LIN {X 0,Y 573.225,Z 559.074,A -85,B 0,C 180,E1 -2028.544,E2 -2028.544} C_VEL
LIN {X 0,Y 573.245,Z 559.083,A -85,B 0,C 180,E1 -2031.3,E2 -2031.3} C_VEL
LIN {X 0,Y 573.262,Z 559.073,A -85,B 0,C 180,E1 -2034.012,E2 -2034.012} C_VEL
LIN {X 0,Y 573.284,Z 559.068,A -85,B 0,C 180,E1 -2036.52,E2 -2036.52} C_VEL
LIN {X 0,Y 573.227,Z 559.08,A -85,B 0,C 180,E1 -2039.119,E2 -2039.119} C_VEL
LIN {X 0,Y 573.238,Z 559.084,A -85,B 0,C 180,E1 -2041.436,E2 -2041.436} C_VEL
LIN {X 0,Y 573.224,Z 559.183,A -85,B 0,C 180,E1 -2043.059,E2 -2043.059} C_VEL
LIN {X 0,Y 573.192,Z 564.644,A -85,B 0,C 180,E1 -2044.24,E2 -2044.24} C_VEL
LIN {X 0,Y 574.076,Z 569.754,A -85,B 0,C 180,E1 -2044.33,E2 -2044.33} C_VEL
LIN {X 0,Y 573.861,Z 670.37,A -85,B 0,C 180,E1 -2045.61,E2 -2045.61} C_VEL
LIN {X 0,Y 573.739,Z 683.395,A -85,B 0,C 180,E1 -2045.918,E2 -2045.918} C_VEL
LIN {X 0,Y 573.708,Z 696.354,A -85,B 0,C 180,E1 -2046.379,E2 -2046.379} C_VEL
LIN {X 0,Y 573.566,Z 707.573,A -85,B 0,C 180,E1 -2046.915,E2 -2046.915} C_VEL
LIN {X 0,Y 573.446,Z 718.445,A -85,B 0,C 180,E1 -2047.576,E2 -2047.576} C_VEL
LIN {X 0,Y 573.349,Z 729.528,A -85,B 0,C 180,E1 -2048.425,E2 -2048.425} C_VEL
LIN {X 0,Y 573.225,Z 739.378,A -85,B 0,C 180,E1 -2049.361,E2 -2049.361} C_VEL
LIN {X 0,Y 573.144,Z 747.345,A -85,B 0,C 180,E1 -2050.294,E2 -2050.294} C_VEL
LIN {X 0,Y 573.076,Z 755.071,A -85,B 0,C 180,E1 -2051.407,E2 -2051.407} C_VEL
LIN {X 0,Y 573.032,Z 761.181,A -85,B 0,C 180,E1 -2052.514,E2 -2052.514} C_VEL
LIN {X 0,Y 572.983,Z 765.933,A -85,B 0,C 180,E1 -2053.614,E2 -2053.614} C_VEL
LIN {X 0,Y 572.982,Z 769.489,A -85,B 0,C 180,E1 -2054.71,E2 -2054.71} C_VEL
LIN {X 0,Y 572.977,Z 771.973,A -85,B 0,C 180,E1 -2055.8,E2 -2055.8} C_VEL
LIN {X 0,Y 572.969,Z 773.055,A -85,B 0,C 180,E1 -2056.523,E2 -2056.523} C_VEL
LIN {X 0,Y 572.947,Z 773.988,A -85,B 0,C 180,E1 -2057.964,E2 -2057.964} C_VEL
LIN {X 0,Y 572.985,Z 773.691,A -85,B 0,C 180,E1 -2058.888,E2 -2058.888} C_VEL
LIN {X 0,Y 572.975,Z 772.265,A -85,B 0,C 180,E1 -2060.112,E2 -2060.112} C_VEL
LIN {X 0,Y 572.932,Z 770.885,A -85,B 0,C 180,E1 -2060.824,E2 -2060.824} C_VEL
LIN {X 0,Y 573.004,Z 767.965,A -85,B 0,C 180,E1 -2061.892,E2 -2061.892} C_VEL
LIN {X 0,Y 573.057,Z 762.966,A -85,B 0,C 180,E1 -2063.193,E2 -2063.193} C_VEL
LIN {X 0,Y 573.079,Z 756.944,A -85,B 0,C 180,E1 -2064.37,E2 -2064.37} C_VEL
LIN {X 0,Y 573.114,Z 750.112,A -85,B 0,C 180,E1 -2065.428,E2 -2065.428} C_VEL
LIN {X 0,Y 573.17,Z 741.607,A -85,B 0,C 180,E1 -2066.485,E2 -2066.485} C_VEL
LIN {X 0,Y 573.292,Z 732.912,A -85,B 0,C 180,E1 -2067.365,E2 -2067.365} C_VEL
LIN {X 0,Y 573.396,Z 722.256,A -85,B 0,C 180,E1 -2068.244,E2 -2068.244} C_VEL
LIN {X 0,Y 573.471,Z 711.617,A -85,B 0,C 180,E1 -2068.947,E2 -2068.947} C_VEL
LIN {X 0,Y 573.664,Z 699.775,A -85,B 0,C 180,E1 -2069.561,E2 -2069.561} C_VEL
LIN {X 0,Y 573.749,Z 687.491,A -85,B 0,C 180,E1 -2070.044,E2 -2070.044} C_VEL
LIN {X 0,Y 573.849,Z 674.654,A -85,B 0,C 180,E1 -2070.395,E2 -2070.395} C_VEL
LIN {X 0,Y 573.921,Z 659.373,A -85,B 0,C 180,E1 -2070.636,E2 -2070.636} C_VEL
LIN {X 0,Y 573.969,Z 568.053,A -85,B 0,C 180,E1 -2071.784,E2 -2071.784} C_VEL
LIN {X 0,Y 573.232,Z 563.728,A -85,B 0,C 180,E1 -2071.866,E2 -2071.866} C_VEL
LIN {X 0,Y 573.305,Z 559.069,A -85,B 0,C 180,E1 -2072.767,E2 -2072.767} C_VEL
LIN {X 0,Y 573.29,Z 559.072,A -85,B 0,C 180,E1 -2075.628,E2 -2075.628} C_VEL
LIN {X 0,Y 573.275,Z 559.075,A -85,B 0,C 180,E1 -2077.75,E2 -2077.75} C_VEL
LIN {X 0,Y 573.266,Z 559.073,A -85,B 0,C 180,E1 -2080.596,E2 -2080.596} C_VEL
LIN {X 0,Y 573.267,Z 559.071,A -85,B 0,C 180,E1 -2082.748,E2 -2082.748} C_VEL
LIN {X 0,Y 573.238,Z 559.074,A -85,B 0,C 180,E1 -2084.919,E2 -2084.919} C_VEL
LIN {X 0,Y 573.252,Z 559.08,A -85,B 0,C 180,E1 -2087.848,E2 -2087.848} C_VEL
LIN {X 0,Y 573.253,Z 559.082,A -85,B 0,C 180,E1 -2090.076,E2 -2090.076} C_VEL
LIN {X 0,Y 573.235,Z 559.074,A -85,B 0,C 180,E1 -2093.099,E2 -2093.099} C_VEL
LIN {X 0,Y 573.255,Z 559.074,A -85,B 0,C 180,E1 -2095.409,E2 -2095.409} C_VEL
LIN {X 0,Y 573.264,Z 559.081,A -85,B 0,C 180,E1 -2098.031,E2 -2098.031} C_VEL
LIN {X 0,Y 573.302,Z 559.069,A -85,B 0,C 180,E1 -2101.193,E2 -2101.193} C_VEL
LIN {X 0,Y 573.274,Z 559.083,A -85,B 0,C 180,E1 -2101.349,E2 -2101.349} C_VEL
LIN {X 0,Y 573.265,Z 563.756,A -85,B 0,C 180,E1 -2102.23,E2 -2102.23} C_VEL
LIN {X 0,Y 574.042,Z 569.524,A -85,B 0,C 180,E1 -2102.326,E2 -2102.326} C_VEL
LIN {X 0,Y 573.844,Z 669.887,A -85,B 0,C 180,E1 -2103.605,E2 -2103.605} C_VEL
LIN {X 0,Y 573.794,Z 682.353,A -85,B 0,C 180,E1 -2103.889,E2 -2103.889} C_VEL
LIN {X 0,Y 573.686,Z 696.565,A -85,B 0,C 180,E1 -2104.388,E2 -2104.388} C_VEL
LIN {X 0,Y 573.581,Z 707.912,A -85,B 0,C 180,E1 -2104.938,E2 -2104.938} C_VEL
LIN {X 0,Y 573.433,Z 718.746,A -85,B 0,C 180,E1 -2105.602,E2 -2105.602} C_VEL
LIN {X 0,Y 573.348,Z 728.828,A -85,B 0,C 180,E1 -2106.367,E2 -2106.367} C_VEL
LIN {X 0,Y 573.254,Z 738.606,A -85,B 0,C 180,E1 -2107.28,E2 -2107.28} C_VEL
LIN {X 0,Y 573.136,Z 747.372,A -85,B 0,C 180,E1 -2108.298,E2 -2108.298} C_VEL
LIN {X 0,Y 573.087,Z 755.074,A -85,B 0,C 180,E1 -2109.412,E2 -2109.412} C_VEL
LIN {X 0,Y 573.036,Z 761.292,A -85,B 0,C 180,E1 -2110.542,E2 -2110.542} C_VEL
LIN {X 0,Y 573.007,Z 765.724,A -85,B 0,C 180,E1 -2111.567,E2 -2111.567} C_VEL
LIN {X 0,Y 572.975,Z 769.189,A -85,B 0,C 180,E1 -2112.612,E2 -2112.612} C_VEL
LIN {X 0,Y 572.925,Z 771.635,A -85,B 0,C 180,E1 -2113.635,E2 -2113.635} C_VEL
LIN {X 0,Y 572.936,Z 773.189,A -85,B 0,C 180,E1 -2114.646,E2 -2114.646} C_VEL
LIN {X 0,Y 572.936,Z 773.902,A -85,B 0,C 180,E1 -2115.637,E2 -2115.637} C_VEL
LIN {X 0,Y 572.929,Z 773.834,A -85,B 0,C 180,E1 -2116.611,E2 -2116.611} C_VEL
LIN {X 0,Y 572.98,Z 773.026,A -85,B 0,C 180,E1 -2117.576,E2 -2117.576} C_VEL
LIN {X 0,Y 572.964,Z 770.494,A -85,B 0,C 180,E1 -2118.987,E2 -2118.987} C_VEL
LIN {X 0,Y 572.988,Z 766.315,A -85,B 0,C 180,E1 -2120.371,E2 -2120.371} C_VEL
LIN {X 0,Y 573.027,Z 761.415,A -85,B 0,C 180,E1 -2121.524,E2 -2121.524} C_VEL
LIN {X 0,Y 573.043,Z 755.909,A -85,B 0,C 180,E1 -2122.542,E2 -2122.542} C_VEL
LIN {X 0,Y 573.112,Z 749.511,A -85,B 0,C 180,E1 -2123.505,E2 -2123.505} C_VEL
LIN {X 0,Y 573.184,Z 742.505,A -85,B 0,C 180,E1 -2124.379,E2 -2124.379} C_VEL
LIN {X 0,Y 573.271,Z 734.419,A -85,B 0,C 180,E1 -2125.222,E2 -2125.222} C_VEL
LIN {X 0,Y 573.383,Z 724.221,A -85,B 0,C 180,E1 -2126.095,E2 -2126.095} C_VEL
LIN {X 0,Y 573.47,Z 713.308,A -85,B 0,C 180,E1 -2126.846,E2 -2126.846} C_VEL
LIN {X 0,Y 573.612,Z 701.541,A -85,B 0,C 180,E1 -2127.477,E2 -2127.477} C_VEL
LIN {X 0,Y 573.704,Z 689.731,A -85,B 0,C 180,E1 -2127.963,E2 -2127.963} C_VEL
LIN {X 0,Y 573.78,Z 677.38,A -85,B 0,C 180,E1 -2128.331,E2 -2128.331} C_VEL
LIN {X 0,Y 573.889,Z 663.987,A -85,B 0,C 180,E1 -2128.579,E2 -2128.579} C_VEL
LIN {X 0,Y 574.001,Z 569.434,A -85,B 0,C 180,E1 -2129.766,E2 -2129.766} C_VEL
LIN {X 0,Y 573.2,Z 564.597,A -85,B 0,C 180,E1 -2129.86,E2 -2129.86} C_VEL
LIN {X 0,Y 573.265,Z 559.076,A -85,B 0,C 180,E1 -2131.086,E2 -2131.086} C_VEL
LIN {X 0,Y 573.281,Z 559.071,A -85,B 0,C 180,E1 -2133.811,E2 -2133.811} C_VEL
LIN {X 0,Y 573.225,Z 559.08,A -85,B 0,C 180,E1 -2136.134,E2 -2136.134} C_VEL
LIN {X 0,Y 573.253,Z 559.074,A -85,B 0,C 180,E1 -2139.174,E2 -2139.174} C_VEL
LIN {X 0,Y 573.231,Z 559.076,A -85,B 0,C 180,E1 -2141.411,E2 -2141.411} C_VEL
LIN {X 0,Y 573.25,Z 559.073,A -85,B 0,C 180,E1 -2143.622,E2 -2143.622} C_VEL
LIN {X 0,Y 573.231,Z 559.085,A -85,B 0,C 180,E1 -2146.529,E2 -2146.529} C_VEL
LIN {X 0,Y 573.273,Z 559.077,A -85,B 0,C 180,E1 -2148.734,E2 -2148.734} C_VEL
LIN {X 0,Y 573.299,Z 559.067,A -85,B 0,C 180,E1 -2151.541,E2 -2151.541} C_VEL
LIN {X 0,Y 573.285,Z 559.076,A -85,B 0,C 180,E1 -2154.372,E2 -2154.372} C_VEL
LIN {X 0,Y 573.306,Z 559.066,A -85,B 0,C 180,E1 -2157.189,E2 -2157.189} C_VEL
LIN {X 0,Y 573.311,Z 559.068,A -85,B 0,C 180,E1 -2160,E2 -2160} C_VEL
LIN {X 0,Y 573.305,Z 559.071,A -85,B 0,C 180,E1 -2162.811,E2 -2162.811} C_VEL
LIN {X 0,Y 573.29,Z 559.068,A -85,B 0,C 180,E1 -2165.628,E2 -2165.628} C_VEL
LIN {X 0,Y 573.299,Z 559.075,A -85,B 0,C 180,E1 -2168.459,E2 -2168.459} C_VEL
LIN {X 0,Y 573.288,Z 559.068,A -85,B 0,C 180,E1 -2171.312,E2 -2171.312} C_VEL
LIN {X 0,Y 573.271,Z 559.077,A -85,B 0,C 180,E1 -2174.425,E2 -2174.425} C_VEL
LIN {X 0,Y 573.251,Z 559.073,A -85,B 0,C 180,E1 -2177.112,E2 -2177.112} C_VEL
LIN {X 0,Y 573.25,Z 559.075,A -85,B 0,C 180,E1 -2180.077,E2 -2180.077} C_VEL
LIN {X 0,Y 573.263,Z 559.072,A -85,B 0,C 180,E1 -2183.154,E2 -2183.154} C_VEL
LIN {X 0,Y 573.282,Z 559.074,A -85,B 0,C 180,E1 -2186.189,E2 -2186.189} C_VEL
LIN {X 0,Y 573.236,Z 559.084,A -85,B 0,C 180,E1 -2188.565,E2 -2188.565} C_VEL
LIN {X 0,Y 573.234,Z 559.077,A -85,B 0,C 180,E1 -2190.993,E2 -2190.993} C_VEL
LIN {X 0,Y 573.281,Z 559.068,A -85,B 0,C 180,E1 -2193.529,E2 -2193.529} C_VEL
LIN {X 0,Y 573.254,Z 559.076,A -85,B 0,C 180,E1 -2196.049,E2 -2196.049} C_VEL
LIN {X 0,Y 573.245,Z 559.08,A -85,B 0,C 180,E1 -2198.702,E2 -2198.702} C_VEL
LIN {X 0,Y 573.249,Z 559.073,A -85,B 0,C 180,E1 -2201.597,E2 -2201.597} C_VEL
LIN {X 0,Y 573.234,Z 559.082,A -85,B 0,C 180,E1 -2204.334,E2 -2204.334} C_VEL
LIN {X 0,Y 573.236,Z 559.075,A -85,B 0,C 180,E1 -2207.359,E2 -2207.359} C_VEL
LIN {X 0,Y 573.244,Z 559.082,A -85,B 0,C 180,E1 -2210.394,E2 -2210.394} C_VEL
LIN {X 0,Y 573.249,Z 559.075,A -85,B 0,C 180,E1 -2213.078,E2 -2213.078} C_VEL
LIN {X 0,Y 573.27,Z 559.071,A -85,B 0,C 180,E1 -2215.673,E2 -2215.673} C_VEL
LIN {X 0,Y 573.24,Z 559.08,A -85,B 0,C 180,E1 -2218.185,E2 -2218.185} C_VEL
LIN {X 0,Y 573.264,Z 559.08,A -85,B 0,C 180,E1 -2220.635,E2 -2220.635} C_VEL
LIN {X 0,Y 573.251,Z 559.077,A -85,B 0,C 180,E1 -2223.025,E2 -2223.025} C_VEL
LIN {X 0,Y 573.267,Z 559.094,A -85,B 0,C 180,E1 -2224.494,E2 -2224.494} C_VEL
LIN {X 0,Y 574.435,Z 565.71,A -85,B 0,C 180,E1 -2225.42,E2 -2225.42} C_VEL
LIN {X 0,Y 574.164,Z 586.292,A -85,B 0,C 180,E1 -2228.079,E2 -2228.079} C_VEL
LIN {X 0,Y 573.878,Z 608.344,A -85,B 0,C 180,E1 -2230.878,E2 -2230.878} C_VEL
LIN {X 0,Y 573.631,Z 631.866,A -85,B 0,C 180,E1 -2233.816,E2 -2233.816} C_VEL
LIN {X 0,Y 573.476,Z 650.794,A -85,B 0,C 180,E1 -2236.152,E2 -2236.152} C_VEL
LIN {X 0,Y 574.051,Z 655.747,A -85,B 0,C 180,E1 -2236.234,E2 -2236.234} C_VEL
LIN {X 0,Y 573.897,Z 759.962,A -85,B 0,C 180,E1 -2237.558,E2 -2237.558} C_VEL
LIN {X 0,Y 573.8,Z 772.463,A -85,B 0,C 180,E1 -2237.848,E2 -2237.848} C_VEL
LIN {X 0,Y 573.701,Z 784.92,A -85,B 0,C 180,E1 -2238.276,E2 -2238.276} C_VEL
LIN {X 0,Y 573.604,Z 795.992,A -85,B 0,C 180,E1 -2238.787,E2 -2238.787} C_VEL
LIN {X 0,Y 573.508,Z 806.59,A -85,B 0,C 180,E1 -2239.408,E2 -2239.408} C_VEL
LIN {X 0,Y 573.356,Z 817.476,A -85,B 0,C 180,E1 -2240.208,E2 -2240.208} C_VEL
LIN {X 0,Y 573.241,Z 828.115,A -85,B 0,C 180,E1 -2241.185,E2 -2241.185} C_VEL
LIN {X 0,Y 573.161,Z 835.962,A -85,B 0,C 180,E1 -2242.071,E2 -2242.071} C_VEL
LIN {X 0,Y 573.072,Z 843.955,A -85,B 0,C 180,E1 -2243.186,E2 -2243.186} C_VEL
LIN {X 0,Y 573.07,Z 850.68,A -85,B 0,C 180,E1 -2244.37,E2 -2244.37} C_VEL
LIN {X 0,Y 573.029,Z 855.372,A -85,B 0,C 180,E1 -2245.428,E2 -2245.428} C_VEL
LIN {X 0,Y 573.023,Z 858.958,A -85,B 0,C 180,E1 -2246.484,E2 -2246.484} C_VEL
LIN {X 0,Y 572.959,Z 860.81,A -85,B 0,C 180,E1 -2247.188,E2 -2247.188} C_VEL
LIN {X 0,Y 572.937,Z 862.2,A -85,B 0,C 180,E1 -2247.891,E2 -2247.891} C_VEL
LIN {X 0,Y 572.941,Z 863.785,A -85,B 0,C 180,E1 -2249.297,E2 -2249.297} C_VEL
LIN {X 0,Y 572.938,Z 864,A -85,B 0,C 180,E1 -2250,E2 -2250} C_VEL
LIN {X 0,Y 572.946,Z 863.185,A -85,B 0,C 180,E1 -2251.406,E2 -2251.406} C_VEL
LIN {X 0,Y 572.937,Z 862.199,A -85,B 0,C 180,E1 -2252.109,E2 -2252.109} C_VEL
LIN {X 0,Y 572.959,Z 860.809,A -85,B 0,C 180,E1 -2252.812,E2 -2252.812} C_VEL
LIN {X 0,Y 573.015,Z 857.896,A -85,B 0,C 180,E1 -2253.868,E2 -2253.868} C_VEL
LIN {X 0,Y 572.963,Z 853.95,A -85,B 0,C 180,E1 -2254.925,E2 -2254.925} C_VEL
LIN {X 0,Y 573.064,Z 847.878,A -85,B 0,C 180,E1 -2256.16,E2 -2256.16} C_VEL
LIN {X 0,Y 573.119,Z 841.239,A -85,B 0,C 180,E1 -2257.221,E2 -2257.221} C_VEL
LIN {X 0,Y 573.201,Z 832.992,A -85,B 0,C 180,E1 -2258.283,E2 -2258.283} C_VEL
LIN {X 0,Y 573.286,Z 824.54,A -85,B 0,C 180,E1 -2259.17,E2 -2259.17} C_VEL
LIN {X 0,Y 573.423,Z 814.1,A -85,B 0,C 180,E1 -2260.058,E2 -2260.058} C_VEL
LIN {X 0,Y 573.549,Z 802.357,A -85,B 0,C 180,E1 -2260.857,E2 -2260.857} C_VEL
LIN {X 0,Y 573.652,Z 791.288,A -85,B 0,C 180,E1 -2261.447,E2 -2261.447} C_VEL
LIN {X 0,Y 573.775,Z 778.188,A -85,B 0,C 180,E1 -2261.973,E2 -2261.973} C_VEL
LIN {X 0,Y 573.823,Z 765.535,A -85,B 0,C 180,E1 -2262.331,E2 -2262.331} C_VEL
LIN {X 0,Y 573.932,Z 752.335,A -85,B 0,C 180,E1 -2262.553,E2 -2262.553} C_VEL
LIN {X 0,Y 573.99,Z 653.289,A -85,B 0,C 180,E1 -2263.799,E2 -2263.799} C_VEL
LIN {X 0,Y 573.542,Z 649.727,A -85,B 0,C 180,E1 -2263.869,E2 -2263.869} C_VEL
LIN {X 0,Y 573.79,Z 623.173,A -85,B 0,C 180,E1 -2266.728,E2 -2266.728} C_VEL
LIN {X 0,Y 574.103,Z 595.953,A -85,B 0,C 180,E1 -2269.699,E2 -2269.699} C_VEL
LIN {X 0,Y 574.439,Z 570.909,A -85,B 0,C 180,E1 -2272.477,E2 -2272.477} C_VEL
LIN {X 0,Y 574.442,Z 564.474,A -85,B 0,C 180,E1 -2273.203,E2 -2273.203} C_VEL
LIN {X 0,Y 573.248,Z 559.083,A -85,B 0,C 180,E1 -2273.888,E2 -2273.888} C_VEL
LIN {X 0,Y 573.27,Z 559.073,A -85,B 0,C 180,E1 -2276.499,E2 -2276.499} C_VEL
LIN {X 0,Y 573.266,Z 559.073,A -85,B 0,C 180,E1 -2279.365,E2 -2279.365} C_VEL
LIN {X 0,Y 573.253,Z 559.078,A -85,B 0,C 180,E1 -2282.228,E2 -2282.228} C_VEL
LIN {X 0,Y 573.25,Z 559.073,A -85,B 0,C 180,E1 -2284.773,E2 -2284.773} C_VEL
LIN {X 0,Y 573.251,Z 559.073,A -85,B 0,C 180,E1 -2287.165,E2 -2287.165} C_VEL
LIN {X 0,Y 573.247,Z 559.076,A -85,B 0,C 180,E1 -2289.606,E2 -2289.606} C_VEL
LIN {X 0,Y 573.238,Z 559.076,A -85,B 0,C 180,E1 -2292.641,E2 -2292.641} C_VEL
LIN {X 0,Y 573.235,Z 559.077,A -85,B 0,C 180,E1 -2295.666,E2 -2295.666} C_VEL
LIN {X 0,Y 573.256,Z 559.076,A -85,B 0,C 180,E1 -2298.545,E2 -2298.545} C_VEL
LIN {X 0,Y 573.246,Z 559.072,A -85,B 0,C 180,E1 -2301.299,E2 -2301.299} C_VEL
LIN {X 0,Y 573.258,Z 559.078,A -85,B 0,C 180,E1 -2304.01,E2 -2304.01} C_VEL
LIN {X 0,Y 573.277,Z 559.075,A -85,B 0,C 180,E1 -2306.518,E2 -2306.518} C_VEL
LIN {X 0,Y 573.236,Z 559.074,A -85,B 0,C 180,E1 -2309.114,E2 -2309.114} C_VEL
LIN {X 0,Y 573.255,Z 559.074,A -85,B 0,C 180,E1 -2311.968,E2 -2311.968} C_VEL
LIN {X 0,Y 573.251,Z 559.079,A -85,B 0,C 180,E1 -2314.59,E2 -2314.59} C_VEL
LIN {X 0,Y 573.228,Z 559.073,A -85,B 0,C 180,E1 -2317.662,E2 -2317.662} C_VEL
LIN {X 0,Y 573.247,Z 559.075,A -85,B 0,C 180,E1 -2319.923,E2 -2319.923} C_VEL
LIN {X 0,Y 573.251,Z 559.073,A -85,B 0,C 180,E1 -2322.989,E2 -2322.989} C_VEL
LIN {X 0,Y 573.262,Z 559.07,A -85,B 0,C 180,E1 -2325.807,E2 -2325.807} C_VEL
LIN {X 0,Y 573.273,Z 559.076,A -85,B 0,C 180,E1 -2328.734,E2 -2328.734} C_VEL
LIN {X 0,Y 573.299,Z 559.064,A -85,B 0,C 180,E1 -2331.541,E2 -2331.541} C_VEL
LIN {X 0,Y 573.292,Z 559.073,A -85,B 0,C 180,E1 -2334.372,E2 -2334.372} C_VEL
LIN {X 0,Y 573.3,Z 559.064,A -85,B 0,C 180,E1 -2337.892,E2 -2337.892} C_VEL
LIN {X 0,Y 573.332,Z 559.071,A -85,B 0,C 180,E1 -2340.702,E2 -2340.702} C_VEL
LIN {X 0,Y 573.232,Z 559.075,A -85,B 0,C 180,E1 -2343.515,E2 -2343.515} C_VEL
LIN {X 0,Y 573.29,Z 559.065,A -85,B 0,C 180,E1 -2345.628,E2 -2345.628} C_VEL
LIN {X 0,Y 573.299,Z 559.07,A -85,B 0,C 180,E1 -2348.459,E2 -2348.459} C_VEL
LIN {X 0,Y 573.288,Z 559.069,A -85,B 0,C 180,E1 -2351.312,E2 -2351.312} C_VEL
LIN {X 0,Y 573.27,Z 559.072,A -85,B 0,C 180,E1 -2354.425,E2 -2354.425} C_VEL
LIN {X 0,Y 573.25,Z 559.079,A -85,B 0,C 180,E1 -2357.112,E2 -2357.112} C_VEL
LIN {X 0,Y 573.247,Z 559.072,A -85,B 0,C 180,E1 -2360.077,E2 -2360.077} C_VEL
LIN {X 0,Y 573.228,Z 559.076,A -85,B 0,C 180,E1 -2362.338,E2 -2362.338} C_VEL
LIN {X 0,Y 573.243,Z 559.073,A -85,B 0,C 180,E1 -2364.403,E2 -2364.403} C_VEL
LIN {X 0,Y 572.618,Z 559.159,A -85,B 0,C 180,E1 -2364.99,E2 -2364.99} C_VEL
LIN {X 0,Y 569.78,Z 559.515,A -85,B 0,C 180,E1 -2365.942,E2 -2365.942} C_VEL
LIN {X 0,Y 567.352,Z 559.817,A -85,B 0,C 180,E1 -2366.708,E2 -2366.708} C_VEL
LIN {X 0,Y 566.299,Z 559.945,A -85,B 0,C 180,E1 -2367.299,E2 -2367.299} C_VEL
LIN {X 0,Y 566.21,Z 559.953,A -85,B 0,C 180,E1 -2367.499,E2 -2367.499} C_VEL
LIN {X 0,Y 566.186,Z 559.953,A -85,B 0,C 180,E1 -2370.593,E2 -2370.593} C_VEL
LIN {X 0,Y 566.221,Z 559.958,A -85,B 0,C 180,E1 -2373.102,E2 -2373.102} C_VEL
LIN {X 0,Y 566.205,Z 559.953,A -85,B 0,C 180,E1 -2375.689,E2 -2375.689} C_VEL
LIN {X 0,Y 566.212,Z 559.951,A -85,B 0,C 180,E1 -2378.56,E2 -2378.56} C_VEL
LIN {X 0,Y 566.206,Z 559.958,A -85,B 0,C 180,E1 -2381.137,E2 -2381.137} C_VEL
LIN {X 0,Y 566.196,Z 559.952,A -85,B 0,C 180,E1 -2384.036,E2 -2384.036} C_VEL
LIN {X 0,Y 566.197,Z 559.957,A -85,B 0,C 180,E1 -2387.084,E2 -2387.084} C_VEL
LIN {X 0,Y 566.223,Z 559.951,A -85,B 0,C 180,E1 -2389.804,E2 -2389.804} C_VEL
LIN {X 0,Y 566.196,Z 559.951,A -85,B 0,C 180,E1 -2392.6,E2 -2392.6} C_VEL
LIN {X 0,Y 566.218,Z 559.955,A -85,B 0,C 180,E1 -2395.184,E2 -2395.184} C_VEL
LIN {X 0,Y 566.23,Z 559.953,A -85,B 0,C 180,E1 -2397.744,E2 -2397.744} C_VEL
LIN {X 0,Y 566.202,Z 559.951,A -85,B 0,C 180,E1 -2400.329,E2 -2400.329} C_VEL
LIN {X 0,Y 566.162,Z 559.979,A -85,B 0,C 180,E1 -2403.042,E2 -2403.042} C_VEL
LIN {X 0,Y 566.147,Z 564.646,A -85,B 0,C 180,E1 -2404.065,E2 -2404.065} C_VEL
LIN {X 0,Y 567.187,Z 571.012,A -85,B 0,C 180,E1 -2404.176,E2 -2404.176} C_VEL
LIN {X 0,Y 566.931,Z 670.77,A -85,B 0,C 180,E1 -2405.463,E2 -2405.463} C_VEL
LIN {X 0,Y 566.787,Z 684.453,A -85,B 0,C 180,E1 -2405.798,E2 -2405.798} C_VEL
LIN {X 0,Y 566.723,Z 697.574,A -85,B 0,C 180,E1 -2406.286,E2 -2406.286} C_VEL
LIN {X 0,Y 566.563,Z 709.826,A -85,B 0,C 180,E1 -2406.903,E2 -2406.903} C_VEL
LIN {X 0,Y 566.396,Z 721.544,A -85,B 0,C 180,E1 -2407.667,E2 -2407.667} C_VEL
LIN {X 0,Y 566.295,Z 730.649,A -85,B 0,C 180,E1 -2408.402,E2 -2408.402} C_VEL
LIN {X 0,Y 566.17,Z 739.654,A -85,B 0,C 180,E1 -2409.282,E2 -2409.282} C_VEL
LIN {X 0,Y 566.07,Z 747.573,A -85,B 0,C 180,E1 -2410.226,E2 -2410.226} C_VEL
LIN {X 0,Y 566.015,Z 755.253,A -85,B 0,C 180,E1 -2411.354,E2 -2411.354} C_VEL
LIN {X 0,Y 565.945,Z 760.404,A -85,B 0,C 180,E1 -2412.288,E2 -2412.288} C_VEL
LIN {X 0,Y 565.92,Z 765.328,A -85,B 0,C 180,E1 -2413.404,E2 -2413.404} C_VEL
LIN {X 0,Y 565.882,Z 769.04,A -85,B 0,C 180,E1 -2414.513,E2 -2414.513} C_VEL
LIN {X 0,Y 565.886,Z 771.695,A -85,B 0,C 180,E1 -2415.632,E2 -2415.632} C_VEL
LIN {X 0,Y 565.864,Z 772.877,A -85,B 0,C 180,E1 -2416.351,E2 -2416.351} C_VEL
LIN {X 0,Y 565.844,Z 773.618,A -85,B 0,C 180,E1 -2417.082,E2 -2417.082} C_VEL
LIN {X 0,Y 565.866,Z 773.955,A -85,B 0,C 180,E1 -2417.811,E2 -2417.811} C_VEL
LIN {X 0,Y 565.902,Z 773.725,A -85,B 0,C 180,E1 -2418.847,E2 -2418.847} C_VEL
LIN {X 0,Y 565.883,Z 772.498,A -85,B 0,C 180,E1 -2419.987,E2 -2419.987} C_VEL
LIN {X 0,Y 565.834,Z 771.195,A -85,B 0,C 180,E1 -2420.708,E2 -2420.708} C_VEL
LIN {X 0,Y 565.896,Z 768.415,A -85,B 0,C 180,E1 -2421.789,E2 -2421.789} C_VEL
LIN {X 0,Y 565.965,Z 764.614,A -85,B 0,C 180,E1 -2422.867,E2 -2422.867} C_VEL
LIN {X 0,Y 565.962,Z 759.702,A -85,B 0,C 180,E1 -2423.941,E2 -2423.941} C_VEL
LIN {X 0,Y 565.993,Z 753.537,A -85,B 0,C 180,E1 -2425.014,E2 -2425.014} C_VEL
LIN {X 0,Y 566.074,Z 745.859,A -85,B 0,C 180,E1 -2426.085,E2 -2426.085} C_VEL
LIN {X 0,Y 566.203,Z 736.315,A -85,B 0,C 180,E1 -2427.154,E2 -2427.154} C_VEL
LIN {X 0,Y 566.332,Z 726.454,A -85,B 0,C 180,E1 -2428.044,E2 -2428.044} C_VEL
LIN {X 0,Y 566.432,Z 715.452,A -85,B 0,C 180,E1 -2428.845,E2 -2428.845} C_VEL
LIN {X 0,Y 566.614,Z 704.679,A -85,B 0,C 180,E1 -2429.467,E2 -2429.467} C_VEL
LIN {X 0,Y 566.743,Z 692.834,A -85,B 0,C 180,E1 -2430,E2 -2430} C_VEL
LIN {X 0,Y 566.83,Z 679.904,A -85,B 0,C 180,E1 -2430.422,E2 -2430.422} C_VEL
LIN {X 0,Y 566.991,Z 667.121,A -85,B 0,C 180,E1 -2430.688,E2 -2430.688} C_VEL
LIN {X 0,Y 567.101,Z 569.002,A -85,B 0,C 180,E1 -2431.942,E2 -2431.942} C_VEL
LIN {X 0,Y 566.24,Z 563.704,A -85,B 0,C 180,E1 -2432.045,E2 -2432.045} C_VEL
LIN {X 0,Y 566.275,Z 559.945,A -85,B 0,C 180,E1 -2432.801,E2 -2432.801} C_VEL
LIN {X 0,Y 566.258,Z 559.949,A -85,B 0,C 180,E1 -2435.698,E2 -2435.698} C_VEL
LIN {X 0,Y 566.209,Z 559.953,A -85,B 0,C 180,E1 -2438.566,E2 -2438.566} C_VEL
LIN {X 0,Y 566.245,Z 559.947,A -85,B 0,C 180,E1 -2441.454,E2 -2441.454} C_VEL
LIN {X 0,Y 566.237,Z 559.949,A -85,B 0,C 180,E1 -2444.506,E2 -2444.506} C_VEL
LIN {X 0,Y 566.204,Z 559.951,A -85,B 0,C 180,E1 -2447.331,E2 -2447.331} C_VEL
LIN {X 0,Y 566.215,Z 559.954,A -85,B 0,C 180,E1 -2450.337,E2 -2450.337} C_VEL
LIN {X 0,Y 566.171,Z 559.955,A -85,B 0,C 180,E1 -2453.281,E2 -2453.281} C_VEL
LIN {X 0,Y 566.214,Z 559.955,A -85,B 0,C 180,E1 -2455.748,E2 -2455.748} C_VEL
LIN {X 0,Y 566.206,Z 559.959,A -85,B 0,C 180,E1 -2458.202,E2 -2458.202} C_VEL
LIN {X 0,Y 566.241,Z 559.959,A -85,B 0,C 180,E1 -2461.33,E2 -2461.33} C_VEL
LIN {X 0,Y 566.211,Z 563.718,A -85,B 0,C 180,E1 -2462.047,E2 -2462.047} C_VEL
LIN {X 0,Y 567.167,Z 570.569,A -85,B 0,C 180,E1 -2462.17,E2 -2462.17} C_VEL
LIN {X 0,Y 566.937,Z 669.927,A -85,B 0,C 180,E1 -2463.452,E2 -2463.452} C_VEL
LIN {X 0,Y 566.864,Z 682.326,A -85,B 0,C 180,E1 -2463.737,E2 -2463.737} C_VEL
LIN {X 0,Y 566.719,Z 696.544,A -85,B 0,C 180,E1 -2464.242,E2 -2464.242} C_VEL
LIN {X 0,Y 566.617,Z 707.698,A -85,B 0,C 180,E1 -2464.788,E2 -2464.788} C_VEL
LIN {X 0,Y 566.474,Z 717.842,A -85,B 0,C 180,E1 -2465.41,E2 -2465.41} C_VEL
LIN {X 0,Y 566.349,Z 726.659,A -85,B 0,C 180,E1 -2466.068,E2 -2466.068} C_VEL
LIN {X 0,Y 566.217,Z 735.915,A -85,B 0,C 180,E1 -2466.9,E2 -2466.9} C_VEL
LIN {X 0,Y 566.109,Z 745.134,A -85,B 0,C 180,E1 -2467.916,E2 -2467.916} C_VEL
LIN {X 0,Y 566.038,Z 753.565,A -85,B 0,C 180,E1 -2469.085,E2 -2469.085} C_VEL
LIN {X 0,Y 565.963,Z 760.021,A -85,B 0,C 180,E1 -2470.219,E2 -2470.219} C_VEL
LIN {X 0,Y 565.923,Z 764.325,A -85,B 0,C 180,E1 -2471.161,E2 -2471.161} C_VEL
LIN {X 0,Y 565.92,Z 767.81,A -85,B 0,C 180,E1 -2472.113,E2 -2472.113} C_VEL
LIN {X 0,Y 565.854,Z 770.534,A -85,B 0,C 180,E1 -2473.086,E2 -2473.086} C_VEL
LIN {X 0,Y 565.858,Z 772.453,A -85,B 0,C 180,E1 -2474.068,E2 -2474.068} C_VEL
LIN {X 0,Y 565.831,Z 773.615,A -85,B 0,C 180,E1 -2475.069,E2 -2475.069} C_VEL
LIN {X 0,Y 565.845,Z 773.997,A -85,B 0,C 180,E1 -2476.084,E2 -2476.084} C_VEL
LIN {X 0,Y 565.853,Z 773.549,A -85,B 0,C 180,E1 -2477.119,E2 -2477.119} C_VEL
LIN {X 0,Y 565.857,Z 772.217,A -85,B 0,C 180,E1 -2478.175,E2 -2478.175} C_VEL
LIN {X 0,Y 565.873,Z 769.931,A -85,B 0,C 180,E1 -2479.252,E2 -2479.252} C_VEL
LIN {X 0,Y 565.907,Z 766.58,A -85,B 0,C 180,E1 -2480.35,E2 -2480.35} C_VEL
LIN {X 0,Y 565.945,Z 761.286,A -85,B 0,C 180,E1 -2481.617,E2 -2481.617} C_VEL
LIN {X 0,Y 565.973,Z 755.88,A -85,B 0,C 180,E1 -2482.627,E2 -2482.627} C_VEL
LIN {X 0,Y 566.061,Z 749.221,A -85,B 0,C 180,E1 -2483.637,E2 -2483.637} C_VEL
LIN {X 0,Y 566.124,Z 742.406,A -85,B 0,C 180,E1 -2484.494,E2 -2484.494} C_VEL
LIN {X 0,Y 566.265,Z 733.731,A -85,B 0,C 180,E1 -2485.402,E2 -2485.402} C_VEL
LIN {X 0,Y 566.367,Z 723.972,A -85,B 0,C 180,E1 -2486.24,E2 -2486.24} C_VEL
LIN {X 0,Y 566.509,Z 712.875,A -85,B 0,C 180,E1 -2487.007,E2 -2487.007} C_VEL
LIN {X 0,Y 566.625,Z 701.416,A -85,B 0,C 180,E1 -2487.625,E2 -2487.625} C_VEL
LIN {X 0,Y 566.749,Z 690.293,A -85,B 0,C 180,E1 -2488.091,E2 -2488.091} C_VEL
LIN {X 0,Y 566.856,Z 678.649,A -85,B 0,C 180,E1 -2488.45,E2 -2488.45} C_VEL
LIN {X 0,Y 566.974,Z 666.54,A -85,B 0,C 180,E1 -2488.695,E2 -2488.695} C_VEL
LIN {X 0,Y 567.084,Z 570.15,A -85,B 0,C 180,E1 -2489.928,E2 -2489.928} C_VEL
LIN {X 0,Y 566.171,Z 564.592,A -85,B 0,C 180,E1 -2490.036,E2 -2490.036} C_VEL
LIN {X 0,Y 566.204,Z 559.956,A -85,B 0,C 180,E1 -2491.075,E2 -2491.075} C_VEL
LIN {X 0,Y 566.239,Z 559.948,A -85,B 0,C 180,E1 -2493.46,E2 -2493.46} C_VEL
LIN {X 0,Y 566.191,Z 559.954,A -85,B 0,C 180,E1 -2495.819,E2 -2495.819} C_VEL
LIN {X 0,Y 566.208,Z 559.955,A -85,B 0,C 180,E1 -2498.902,E2 -2498.902} C_VEL
LIN {X 0,Y 566.205,Z 559.952,A -85,B 0,C 180,E1 -2501.172,E2 -2501.172} C_VEL
LIN {X 0,Y 566.212,Z 559.95,A -85,B 0,C 180,E1 -2503.412,E2 -2503.412} C_VEL
LIN {X 0,Y 566.193,Z 559.96,A -85,B 0,C 180,E1 -2506.359,E2 -2506.359} C_VEL
LIN {X 0,Y 566.265,Z 559.951,A -85,B 0,C 180,E1 -2508.654,E2 -2508.654} C_VEL
LIN {X 0,Y 566.241,Z 559.946,A -85,B 0,C 180,E1 -2511.434,E2 -2511.434} C_VEL
LIN {X 0,Y 566.253,Z 559.951,A -85,B 0,C 180,E1 -2514.302,E2 -2514.302} C_VEL
LIN {X 0,Y 566.271,Z 559.943,A -85,B 0,C 180,E1 -2517.866,E2 -2517.866} C_VEL
LIN {X 0,Y 566.298,Z 559.946,A -85,B 0,C 180,E1 -2520.711,E2 -2520.711} C_VEL
LIN {X 0,Y 566.27,Z 559.946,A -85,B 0,C 180,E1 -2522.846,E2 -2522.846} C_VEL
LIN {X 0,Y 566.258,Z 559.944,A -85,B 0,C 180,E1 -2525.698,E2 -2525.698} C_VEL
LIN {X 0,Y 566.241,Z 559.955,A -85,B 0,C 180,E1 -2528.566,E2 -2528.566} C_VEL
LIN {X 0,Y 566.241,Z 559.945,A -85,B 0,C 180,E1 -2531.454,E2 -2531.454} C_VEL
LIN {X 0,Y 566.224,Z 559.956,A -85,B 0,C 180,E1 -2534.507,E2 -2534.507} C_VEL
LIN {X 0,Y 566.195,Z 559.95,A -85,B 0,C 180,E1 -2537.332,E2 -2537.332} C_VEL
LIN {X 0,Y 566.213,Z 559.956,A -85,B 0,C 180,E1 -2540.337,E2 -2540.337} C_VEL
LIN {X 0,Y 566.222,Z 559.947,A -85,B 0,C 180,E1 -2543.403,E2 -2543.403} C_VEL
LIN {X 0,Y 566.218,Z 559.949,A -85,B 0,C 180,E1 -2545.749,E2 -2545.749} C_VEL
LIN {X 0,Y 566.2,Z 559.955,A -85,B 0,C 180,E1 -2548.204,E2 -2548.204} C_VEL
LIN {X 0,Y 566.188,Z 559.961,A -85,B 0,C 180,E1 -2550.592,E2 -2550.592} C_VEL
LIN {X 0,Y 566.222,Z 559.949,A -85,B 0,C 180,E1 -2553.102,E2 -2553.102} C_VEL
LIN {X 0,Y 566.205,Z 559.951,A -85,B 0,C 180,E1 -2555.689,E2 -2555.689} C_VEL
LIN {X 0,Y 566.212,Z 559.958,A -85,B 0,C 180,E1 -2558.56,E2 -2558.56} C_VEL
LIN {X 0,Y 566.207,Z 559.951,A -85,B 0,C 180,E1 -2561.137,E2 -2561.137} C_VEL
LIN {X 0,Y 566.196,Z 559.955,A -85,B 0,C 180,E1 -2564.036,E2 -2564.036} C_VEL
LIN {X 0,Y 566.197,Z 559.954,A -85,B 0,C 180,E1 -2567.084,E2 -2567.084} C_VEL
LIN {X 0,Y 566.224,Z 559.949,A -85,B 0,C 180,E1 -2569.804,E2 -2569.804} C_VEL
LIN {X 0,Y 566.195,Z 559.96,A -85,B 0,C 180,E1 -2572.6,E2 -2572.6} C_VEL
LIN {X 0,Y 566.211,Z 559.951,A -85,B 0,C 180,E1 -2575.183,E2 -2575.183} C_VEL
LIN {X 0,Y 566.23,Z 559.949,A -85,B 0,C 180,E1 -2577.744,E2 -2577.744} C_VEL
LIN {X 0,Y 566.203,Z 559.959,A -85,B 0,C 180,E1 -2580.329,E2 -2580.329} C_VEL
LIN {X 0,Y 566.212,Z 559.959,A -85,B 0,C 180,E1 -2582.662,E2 -2582.662} C_VEL
LIN {X 0,Y 566.236,Z 560.112,A -85,B 0,C 180,E1 -2584.32,E2 -2584.32} C_VEL
LIN {X 0,Y 567.599,Z 567.18,A -85,B 0,C 180,E1 -2585.299,E2 -2585.299} C_VEL
LIN {X 0,Y 567.333,Z 586.292,A -85,B 0,C 180,E1 -2587.801,E2 -2587.801} C_VEL
LIN {X 0,Y 566.953,Z 608.344,A -85,B 0,C 180,E1 -2590.635,E2 -2590.635} C_VEL
LIN {X 0,Y 566.701,Z 629.101,A -85,B 0,C 180,E1 -2593.264,E2 -2593.264} C_VEL
LIN {X 0,Y 566.493,Z 650.794,A -85,B 0,C 180,E1 -2595.978,E2 -2595.978} C_VEL
LIN {X 0,Y 567.203,Z 657.536,A -85,B 0,C 180,E1 -2596.087,E2 -2596.087} C_VEL
LIN {X 0,Y 566.965,Z 759.961,A -85,B 0,C 180,E1 -2597.404,E2 -2597.404} C_VEL
LIN {X 0,Y 566.84,Z 772.462,A -85,B 0,C 180,E1 -2597.696,E2 -2597.696} C_VEL
LIN {X 0,Y 566.752,Z 784.921,A -85,B 0,C 180,E1 -2598.13,E2 -2598.13} C_VEL
LIN {X 0,Y 566.625,Z 797.159,A -85,B 0,C 180,E1 -2598.708,E2 -2598.708} C_VEL
LIN {X 0,Y 566.449,Z 809.206,A -85,B 0,C 180,E1 -2599.455,E2 -2599.455} C_VEL
LIN {X 0,Y 566.319,Z 819.603,A -85,B 0,C 180,E1 -2600.266,E2 -2600.266} C_VEL
LIN {X 0,Y 566.207,Z 828.115,A -85,B 0,C 180,E1 -2601.074,E2 -2601.074} C_VEL
LIN {X 0,Y 566.112,Z 835.962,A -85,B 0,C 180,E1 -2601.972,E2 -2601.972} C_VEL
LIN {X 0,Y 566.003,Z 843.623,A -85,B 0,C 180,E1 -2603.047,E2 -2603.047} C_VEL
LIN {X 0,Y 566.004,Z 850.68,A -85,B 0,C 180,E1 -2604.299,E2 -2604.299} C_VEL
LIN {X 0,Y 565.933,Z 855.372,A -85,B 0,C 180,E1 -2605.37,E2 -2605.37} C_VEL
LIN {X 0,Y 565.927,Z 858.959,A -85,B 0,C 180,E1 -2606.44,E2 -2606.44} C_VEL
LIN {X 0,Y 565.878,Z 860.81,A -85,B 0,C 180,E1 -2607.153,E2 -2607.153} C_VEL
LIN {X 0,Y 565.846,Z 863.186,A -85,B 0,C 180,E1 -2608.577,E2 -2608.577} C_VEL
LIN {X 0,Y 565.839,Z 864,A -85,B 0,C 180,E1 -2610,E2 -2610} C_VEL
LIN {X 0,Y 565.846,Z 863.186,A -85,B 0,C 180,E1 -2611.423,E2 -2611.423} C_VEL
LIN {X 0,Y 565.878,Z 860.808,A -85,B 0,C 180,E1 -2612.847,E2 -2612.847} C_VEL
LIN {X 0,Y 565.926,Z 857.896,A -85,B 0,C 180,E1 -2613.916,E2 -2613.916} C_VEL
LIN {X 0,Y 565.878,Z 853.95,A -85,B 0,C 180,E1 -2614.987,E2 -2614.987} C_VEL
LIN {X 0,Y 566.002,Z 848.868,A -85,B 0,C 180,E1 -2616.058,E2 -2616.058} C_VEL
LIN {X 0,Y 566.04,Z 842.469,A -85,B 0,C 180,E1 -2617.132,E2 -2617.132} C_VEL
LIN {X 0,Y 566.133,Z 834.48,A -85,B 0,C 180,E1 -2618.207,E2 -2618.207} C_VEL
LIN {X 0,Y 566.228,Z 826.338,A -85,B 0,C 180,E1 -2619.105,E2 -2619.105} C_VEL
LIN {X 0,Y 566.343,Z 816.405,A -85,B 0,C 180,E1 -2620.005,E2 -2620.005} C_VEL
LIN {X 0,Y 566.524,Z 805.291,A -85,B 0,C 180,E1 -2620.807,E2 -2620.807} C_VEL
LIN {X 0,Y 566.612,Z 794.182,A -85,B 0,C 180,E1 -2621.446,E2 -2621.446} C_VEL
LIN {X 0,Y 566.76,Z 781.998,A -85,B 0,C 180,E1 -2621.987,E2 -2621.987} C_VEL
LIN {X 0,Y 566.902,Z 769.195,A -85,B 0,C 180,E1 -2622.393,E2 -2622.393} C_VEL
LIN {X 0,Y 566.989,Z 757.128,A -85,B 0,C 180,E1 -2622.641,E2 -2622.641} C_VEL
LIN {X 0,Y 567.104,Z 653.957,A -85,B 0,C 180,E1 -2623.961,E2 -2623.961} C_VEL
LIN {X 0,Y 566.554,Z 649.727,A -85,B 0,C 180,E1 -2624.044,E2 -2624.044} C_VEL
LIN {X 0,Y 566.84,Z 623.355,A -85,B 0,C 180,E1 -2626.919,E2 -2626.919} C_VEL
LIN {X 0,Y 567.212,Z 596.535,A -85,B 0,C 180,E1 -2629.883,E2 -2629.883} C_VEL
LIN {X 0,Y 567.605,Z 572.595,A -85,B 0,C 180,E1 -2632.571,E2 -2632.571} C_VEL
LIN {X 0,Y 567.547,Z 565.852,A -85,B 0,C 180,E1 -2633.344,E2 -2633.344} C_VEL
LIN {X 0,Y 566.226,Z 559.957,A -85,B 0,C 180,E1 -2634.084,E2 -2634.084} C_VEL
LIN {X 0,Y 566.235,Z 559.949,A -85,B 0,C 180,E1 -2636.664,E2 -2636.664} C_VEL
LIN {X 0,Y 566.194,Z 559.952,A -85,B 0,C 180,E1 -2638.952,E2 -2638.952} C_VEL
LIN {X 0,Y 566.196,Z 559.954,A -85,B 0,C 180,E1 -2641.421,E2 -2641.421} C_VEL
LIN {X 0,Y 566.222,Z 559.958,A -85,B 0,C 180,E1 -2643.954,E2 -2643.954} C_VEL
LIN {X 0,Y 566.214,Z 559.951,A -85,B 0,C 180,E1 -2646.568,E2 -2646.568} C_VEL
LIN {X 0,Y 566.212,Z 559.953,A -85,B 0,C 180,E1 -2649.685,E2 -2649.685} C_VEL
LIN {X 0,Y 566.21,Z 559.958,A -85,B 0,C 180,E1 -2652.086,E2 -2652.086} C_VEL
LIN {X 0,Y 566.169,Z 559.954,A -85,B 0,C 180,E1 -2655.035,E2 -2655.035} C_VEL
LIN {X 0,Y 566.22,Z 559.958,A -85,B 0,C 180,E1 -2658.134,E2 -2658.134} C_VEL
LIN {X 0,Y 566.219,Z 559.95,A -85,B 0,C 180,E1 -2660.727,E2 -2660.727} C_VEL
LIN {X 0,Y 566.211,Z 559.952,A -85,B 0,C 180,E1 -2663.783,E2 -2663.783} C_VEL
LIN {X 0,Y 566.204,Z 559.958,A -85,B 0,C 180,E1 -2666.265,E2 -2666.265} C_VEL
LIN {X 0,Y 566.195,Z 559.952,A -85,B 0,C 180,E1 -2668.921,E2 -2668.921} C_VEL
LIN {X 0,Y 566.188,Z 559.951,A -85,B 0,C 180,E1 -2671.046,E2 -2671.046} C_VEL
LIN {X 0,Y 566.239,Z 559.946,A -85,B 0,C 180,E1 -2673.46,E2 -2673.46} C_VEL
LIN {X 0,Y 566.191,Z 559.953,A -85,B 0,C 180,E1 -2675.819,E2 -2675.819} C_VEL
LIN {X 0,Y 566.207,Z 559.952,A -85,B 0,C 180,E1 -2678.902,E2 -2678.902} C_VEL
LIN {X 0,Y 566.204,Z 559.951,A -85,B 0,C 180,E1 -2681.172,E2 -2681.172} C_VEL
LIN {X 0,Y 566.21,Z 559.947,A -85,B 0,C 180,E1 -2683.412,E2 -2683.412} C_VEL
LIN {X 0,Y 566.19,Z 559.958,A -85,B 0,C 180,E1 -2686.359,E2 -2686.359} C_VEL
LIN {X 0,Y 566.265,Z 559.951,A -85,B 0,C 180,E1 -2688.654,E2 -2688.654} C_VEL
LIN {X 0,Y 566.239,Z 559.943,A -85,B 0,C 180,E1 -2691.434,E2 -2691.434} C_VEL
LIN {X 0,Y 566.26,Z 559.948,A -85,B 0,C 180,E1 -2694.302,E2 -2694.302} C_VEL
LIN {X 0,Y 566.271,Z 559.94,A -85,B 0,C 180,E1 -2697.866,E2 -2697.866} C_VEL
LIN {X 0,Y 566.301,Z 559.947,A -85,B 0,C 180,E1 -2700.711,E2 -2700.711} C_VEL
LIN {X 0,Y 566.271,Z 559.95,A -85,B 0,C 180,E1 -2702.846,E2 -2702.846} C_VEL
LIN {X 0,Y 566.258,Z 559.94,A -85,B 0,C 180,E1 -2705.698,E2 -2705.698} C_VEL
LIN {X 0,Y 566.24,Z 559.951,A -85,B 0,C 180,E1 -2708.566,E2 -2708.566} C_VEL
LIN {X 0,Y 566.241,Z 559.945,A -85,B 0,C 180,E1 -2711.454,E2 -2711.454} C_VEL
LIN {X 0,Y 566.223,Z 559.951,A -85,B 0,C 180,E1 -2714.507,E2 -2714.507} C_VEL
LIN {X 0,Y 566.194,Z 559.954,A -85,B 0,C 180,E1 -2717.332,E2 -2717.332} C_VEL
LIN {X 0,Y 566.21,Z 559.95,A -85,B 0,C 180,E1 -2720.337,E2 -2720.337} C_VEL
LIN {X 0,Y 566.181,Z 559.956,A -85,B 0,C 180,E1 -2723.404,E2 -2723.404} C_VEL
LIN {X 0,Y 566.217,Z 559.949,A -85,B 0,C 180,E1 -2725.749,E2 -2725.749} C_VEL
LIN {X 0,Y 566.21,Z 559.953,A -85,B 0,C 180,E1 -2727.499,E2 -2727.499} C_VEL
LIN {X 0,Y 565.531,Z 560.036,A -85,B 0,C 180,E1 -2728.093,E2 -2728.093} C_VEL
LIN {X 0,Y 562.665,Z 560.4,A -85,B 0,C 180,E1 -2729.057,E2 -2729.057} C_VEL
LIN {X 0,Y 560.254,Z 560.694,A -85,B 0,C 180,E1 -2729.832,E2 -2729.832} C_VEL
LIN {X 0,Y 559.226,Z 560.819,A -85,B 0,C 180,E1 -2730.431,E2 -2730.431} C_VEL
LIN {X 0,Y 559.145,Z 560.831,A -85,B 0,C 180,E1 -2730.634,E2 -2730.634} C_VEL
LIN {X 0,Y 559.157,Z 560.83,A -85,B 0,C 180,E1 -2733.575,E2 -2733.575} C_VEL
LIN {X 0,Y 559.162,Z 560.828,A -85,B 0,C 180,E1 -2736.449,E2 -2736.449} C_VEL
LIN {X 0,Y 559.173,Z 560.832,A -85,B 0,C 180,E1 -2738.934,E2 -2738.934} C_VEL
LIN {X 0,Y 559.186,Z 560.822,A -85,B 0,C 180,E1 -2741.768,E2 -2741.768} C_VEL
LIN {X 0,Y 559.135,Z 560.833,A -85,B 0,C 180,E1 -2744.74,E2 -2744.74} C_VEL
LIN {X 0,Y 559.153,Z 560.836,A -85,B 0,C 180,E1 -2747.257,E2 -2747.257} C_VEL
LIN {X 0,Y 559.182,Z 560.826,A -85,B 0,C 180,E1 -2750.136,E2 -2750.136} C_VEL
LIN {X 0,Y 559.144,Z 560.831,A -85,B 0,C 180,E1 -2752.893,E2 -2752.893} C_VEL
LIN {X 0,Y 559.155,Z 560.837,A -85,B 0,C 180,E1 -2755.557,E2 -2755.557} C_VEL
LIN {X 0,Y 559.165,Z 560.829,A -85,B 0,C 180,E1 -2758.138,E2 -2758.138} C_VEL
LIN {X 0,Y 559.142,Z 560.831,A -85,B 0,C 180,E1 -2760.647,E2 -2760.647} C_VEL
LIN {X 0,Y 559.118,Z 560.862,A -85,B 0,C 180,E1 -2763.045,E2 -2763.045} C_VEL
LIN {X 0,Y 559.127,Z 564.816,A -85,B 0,C 180,E1 -2763.892,E2 -2763.892} C_VEL
LIN {X 0,Y 560.278,Z 571.265,A -85,B 0,C 180,E1 -2764.005,E2 -2764.005} C_VEL
LIN {X 0,Y 560.013,Z 669.829,A -85,B 0,C 180,E1 -2765.288,E2 -2765.288} C_VEL
LIN {X 0,Y 559.877,Z 683.1,A -85,B 0,C 180,E1 -2765.603,E2 -2765.603} C_VEL
LIN {X 0,Y 559.783,Z 695.928,A -85,B 0,C 180,E1 -2766.067,E2 -2766.067} C_VEL
LIN {X 0,Y 559.623,Z 707.924,A -85,B 0,C 180,E1 -2766.654,E2 -2766.654} C_VEL
LIN {X 0,Y 559.445,Z 719.323,A -85,B 0,C 180,E1 -2767.374,E2 -2767.374} C_VEL
LIN {X 0,Y 559.297,Z 729.637,A -85,B 0,C 180,E1 -2768.191,E2 -2768.191} C_VEL
LIN {X 0,Y 559.137,Z 739.933,A -85,B 0,C 180,E1 -2769.202,E2 -2769.202} C_VEL
LIN {X 0,Y 559.021,Z 747.806,A -85,B 0,C 180,E1 -2770.158,E2 -2770.158} C_VEL
LIN {X 0,Y 558.941,Z 755.434,A -85,B 0,C 180,E1 -2771.299,E2 -2771.299} C_VEL
LIN {X 0,Y 558.869,Z 761.475,A -85,B 0,C 180,E1 -2772.434,E2 -2772.434} C_VEL
LIN {X 0,Y 558.834,Z 766.155,A -85,B 0,C 180,E1 -2773.563,E2 -2773.563} C_VEL
LIN {X 0,Y 558.776,Z 769.646,A -85,B 0,C 180,E1 -2774.685,E2 -2774.685} C_VEL
LIN {X 0,Y 558.779,Z 771.638,A -85,B 0,C 180,E1 -2775.573,E2 -2775.573} C_VEL
LIN {X 0,Y 558.744,Z 773.513,A -85,B 0,C 180,E1 -2776.915,E2 -2776.915} C_VEL
LIN {X 0,Y 558.771,Z 773.921,A -85,B 0,C 180,E1 -2777.654,E2 -2777.654} C_VEL
LIN {X 0,Y 558.793,Z 773.549,A -85,B 0,C 180,E1 -2779.126,E2 -2779.126} C_VEL
LIN {X 0,Y 558.78,Z 772.732,A -85,B 0,C 180,E1 -2779.859,E2 -2779.859} C_VEL
LIN {X 0,Y 558.745,Z 771.497,A -85,B 0,C 180,E1 -2780.589,E2 -2780.589} C_VEL
LIN {X 0,Y 558.79,Z 768.86,A -85,B 0,C 180,E1 -2781.684,E2 -2781.684} C_VEL
LIN {X 0,Y 558.885,Z 765.206,A -85,B 0,C 180,E1 -2782.776,E2 -2782.776} C_VEL
LIN {X 0,Y 558.885,Z 760.458,A -85,B 0,C 180,E1 -2783.864,E2 -2783.864} C_VEL
LIN {X 0,Y 558.952,Z 753.355,A -85,B 0,C 180,E1 -2785.131,E2 -2785.131} C_VEL
LIN {X 0,Y 559.001,Z 745.63,A -85,B 0,C 180,E1 -2786.216,E2 -2786.216} C_VEL
LIN {X 0,Y 559.169,Z 736.036,A -85,B 0,C 180,E1 -2787.299,E2 -2787.299} C_VEL
LIN {X 0,Y 559.31,Z 726.096,A -85,B 0,C 180,E1 -2788.2,E2 -2788.2} C_VEL
LIN {X 0,Y 559.435,Z 715.013,A -85,B 0,C 180,E1 -2789.01,E2 -2789.01} C_VEL
LIN {X 0,Y 559.679,Z 704.116,A -85,B 0,C 180,E1 -2789.64,E2 -2789.64} C_VEL
LIN {X 0,Y 559.827,Z 692.044,A -85,B 0,C 180,E1 -2790.18,E2 -2790.18} C_VEL
LIN {X 0,Y 559.917,Z 678.81,A -85,B 0,C 180,E1 -2790.607,E2 -2790.607} C_VEL
LIN {X 0,Y 560.062,Z 665.165,A -85,B 0,C 180,E1 -2790.876,E2 -2790.876} C_VEL
LIN {X 0,Y 560.158,Z 569.434,A -85,B 0,C 180,E1 -2792.112,E2 -2792.112} C_VEL
LIN {X 0,Y 559.227,Z 563.683,A -85,B 0,C 180,E1 -2792.228,E2 -2792.228} C_VEL
LIN {X 0,Y 559.224,Z 560.824,A -85,B 0,C 180,E1 -2792.791,E2 -2792.791} C_VEL
LIN {X 0,Y 559.228,Z 560.826,A -85,B 0,C 180,E1 -2795.77,E2 -2795.77} C_VEL
LIN {X 0,Y 559.173,Z 560.828,A -85,B 0,C 180,E1 -2798.674,E2 -2798.674} C_VEL
LIN {X 0,Y 559.209,Z 560.825,A -85,B 0,C 180,E1 -2801.6,E2 -2801.6} C_VEL
LIN {X 0,Y 559.203,Z 560.825,A -85,B 0,C 180,E1 -2804.595,E2 -2804.595} C_VEL
LIN {X 0,Y 559.163,Z 560.831,A -85,B 0,C 180,E1 -2807.556,E2 -2807.556} C_VEL
LIN {X 0,Y 559.171,Z 560.833,A -85,B 0,C 180,E1 -2809.837,E2 -2809.837} C_VEL
LIN {X 0,Y 559.143,Z 560.838,A -85,B 0,C 180,E1 -2812.152,E2 -2812.152} C_VEL
LIN {X 0,Y 559.176,Z 560.827,A -85,B 0,C 180,E1 -2815.297,E2 -2815.297} C_VEL
LIN {X 0,Y 559.192,Z 560.83,A -85,B 0,C 180,E1 -2817.711,E2 -2817.711} C_VEL
LIN {X 0,Y 559.19,Z 560.828,A -85,B 0,C 180,E1 -2821.016,E2 -2821.016} C_VEL
LIN {X 0,Y 559.173,Z 560.929,A -85,B 0,C 180,E1 -2821.327,E2 -2821.327} C_VEL
LIN {X 0,Y 559.162,Z 563.693,A -85,B 0,C 180,E1 -2821.862,E2 -2821.862} C_VEL
LIN {X 0,Y 560.275,Z 571.139,A -85,B 0,C 180,E1 -2822.003,E2 -2822.003} C_VEL
LIN {X 0,Y 560.04,Z 669.536,A -85,B 0,C 180,E1 -2823.288,E2 -2823.288} C_VEL
LIN {X 0,Y 559.922,Z 680.871,A -85,B 0,C 180,E1 -2823.544,E2 -2823.544} C_VEL
LIN {X 0,Y 559.795,Z 693.658,A -85,B 0,C 180,E1 -2823.972,E2 -2823.972} C_VEL
LIN {X 0,Y 559.671,Z 705.387,A -85,B 0,C 180,E1 -2824.516,E2 -2824.516} C_VEL
LIN {X 0,Y 559.485,Z 716.716,A -85,B 0,C 180,E1 -2825.198,E2 -2825.198} C_VEL
LIN {X 0,Y 559.33,Z 725.695,A -85,B 0,C 180,E1 -2825.862,E2 -2825.862} C_VEL
LIN {X 0,Y 559.237,Z 733.796,A -85,B 0,C 180,E1 -2826.577,E2 -2826.577} C_VEL
LIN {X 0,Y 559.121,Z 741.369,A -85,B 0,C 180,E1 -2827.369,E2 -2827.369} C_VEL
LIN {X 0,Y 558.959,Z 749.578,A -85,B 0,C 180,E1 -2828.407,E2 -2828.407} C_VEL
LIN {X 0,Y 558.941,Z 756.096,A -85,B 0,C 180,E1 -2829.417,E2 -2829.417} C_VEL
LIN {X 0,Y 558.864,Z 762.231,A -85,B 0,C 180,E1 -2830.599,E2 -2830.599} C_VEL
LIN {X 0,Y 558.825,Z 766.975,A -85,B 0,C 180,E1 -2831.8,E2 -2831.8} C_VEL
LIN {X 0,Y 558.767,Z 770.752,A -85,B 0,C 180,E1 -2833.155,E2 -2833.155} C_VEL
LIN {X 0,Y 558.77,Z 772.665,A -85,B 0,C 180,E1 -2834.199,E2 -2834.199} C_VEL
LIN {X 0,Y 558.749,Z 773.718,A -85,B 0,C 180,E1 -2835.221,E2 -2835.221} C_VEL
LIN {X 0,Y 558.754,Z 773.967,A -85,B 0,C 180,E1 -2836.228,E2 -2836.228} C_VEL
LIN {X 0,Y 558.749,Z 773.472,A -85,B 0,C 180,E1 -2837.217,E2 -2837.217} C_VEL
LIN {X 0,Y 558.761,Z 772.232,A -85,B 0,C 180,E1 -2838.193,E2 -2838.193} C_VEL
LIN {X 0,Y 558.785,Z 770.271,A -85,B 0,C 180,E1 -2839.155,E2 -2839.155} C_VEL
LIN {X 0,Y 558.8,Z 765.975,A -85,B 0,C 180,E1 -2840.57,E2 -2840.57} C_VEL
LIN {X 0,Y 558.867,Z 761.732,A -85,B 0,C 180,E1 -2841.596,E2 -2841.596} C_VEL
LIN {X 0,Y 558.903,Z 756.339,A -85,B 0,C 180,E1 -2842.633,E2 -2842.633} C_VEL
LIN {X 0,Y 558.992,Z 750.358,A -85,B 0,C 180,E1 -2843.574,E2 -2843.574} C_VEL
LIN {X 0,Y 559.081,Z 743.679,A -85,B 0,C 180,E1 -2844.451,E2 -2844.451} C_VEL
LIN {X 0,Y 559.212,Z 735.541,A -85,B 0,C 180,E1 -2845.341,E2 -2845.341} C_VEL
LIN {X 0,Y 559.332,Z 726.895,A -85,B 0,C 180,E1 -2846.128,E2 -2846.128} C_VEL
LIN {X 0,Y 559.451,Z 718.038,A -85,B 0,C 180,E1 -2846.8,E2 -2846.8} C_VEL
LIN {X 0,Y 559.594,Z 708.114,A -85,B 0,C 180,E1 -2847.42,E2 -2847.42} C_VEL
LIN {X 0,Y 559.774,Z 697.23,A -85,B 0,C 180,E1 -2847.964,E2 -2847.964} C_VEL
LIN {X 0,Y 559.894,Z 683.565,A -85,B 0,C 180,E1 -2848.472,E2 -2848.472} C_VEL
LIN {X 0,Y 560.003,Z 671.035,A -85,B 0,C 180,E1 -2848.776,E2 -2848.776} C_VEL
LIN {X 0,Y 560.118,Z 640.337,A -85,B 0,C 180,E1 -2849.197,E2 -2849.197} C_VEL
LIN {X 0,Y 560.231,Z 571.23,A -85,B 0,C 180,E1 -2850.087,E2 -2850.087} C_VEL
LIN {X 0,Y 559.112,Z 564.613,A -85,B 0,C 180,E1 -2850.212,E2 -2850.212} C_VEL
LIN {X 0,Y 559.153,Z 560.835,A -85,B 0,C 180,E1 -2851.059,E2 -2851.059} C_VEL
LIN {X 0,Y 559.174,Z 560.83,A -85,B 0,C 180,E1 -2853.169,E2 -2853.169} C_VEL
LIN {X 0,Y 559.148,Z 560.831,A -85,B 0,C 180,E1 -2855.494,E2 -2855.494} C_VEL
LIN {X 0,Y 559.169,Z 560.837,A -85,B 0,C 180,E1 -2858.624,E2 -2858.624} C_VEL
LIN {X 0,Y 559.163,Z 560.832,A -85,B 0,C 180,E1 -2860.926,E2 -2860.926} C_VEL
LIN {X 0,Y 559.162,Z 560.83,A -85,B 0,C 180,E1 -2863.948,E2 -2863.948} C_VEL
LIN {X 0,Y 559.166,Z 560.832,A -85,B 0,C 180,E1 -2866.184,E2 -2866.184} C_VEL
LIN {X 0,Y 559.202,Z 560.825,A -85,B 0,C 180,E1 -2869.134,E2 -2869.134} C_VEL
LIN {X 0,Y 559.204,Z 560.826,A -85,B 0,C 180,E1 -2872.054,E2 -2872.054} C_VEL
LIN {X 0,Y 559.253,Z 560.82,A -85,B 0,C 180,E1 -2874.953,E2 -2874.953} C_VEL
LIN {X 0,Y 559.242,Z 560.818,A -85,B 0,C 180,E1 -2877.839,E2 -2877.839} C_VEL
LIN {X 0,Y 559.267,Z 560.822,A -85,B 0,C 180,E1 -2880.72,E2 -2880.72} C_VEL
LIN {X 0,Y 559.236,Z 560.822,A -85,B 0,C 180,E1 -2882.881,E2 -2882.881} C_VEL
LIN {X 0,Y 559.228,Z 560.82,A -85,B 0,C 180,E1 -2885.77,E2 -2885.77} C_VEL
LIN {X 0,Y 559.195,Z 560.83,A -85,B 0,C 180,E1 -2888.674,E2 -2888.674} C_VEL
LIN {X 0,Y 559.199,Z 560.822,A -85,B 0,C 180,E1 -2891.601,E2 -2891.601} C_VEL
LIN {X 0,Y 559.189,Z 560.832,A -85,B 0,C 180,E1 -2894.596,E2 -2894.596} C_VEL
LIN {X 0,Y 559.155,Z 560.827,A -85,B 0,C 180,E1 -2897.557,E2 -2897.557} C_VEL
LIN {X 0,Y 559.167,Z 560.827,A -85,B 0,C 180,E1 -2899.838,E2 -2899.838} C_VEL
LIN {X 0,Y 559.147,Z 560.833,A -85,B 0,C 180,E1 -2902.153,E2 -2902.153} C_VEL
LIN {X 0,Y 559.153,Z 560.837,A -85,B 0,C 180,E1 -2904.505,E2 -2904.505} C_VEL
LIN {X 0,Y 559.172,Z 560.829,A -85,B 0,C 180,E1 -2906.902,E2 -2906.902} C_VEL
LIN {X 0,Y 559.182,Z 560.827,A -85,B 0,C 180,E1 -2909.866,E2 -2909.866} C_VEL
LIN {X 0,Y 559.169,Z 560.833,A -85,B 0,C 180,E1 -2912.715,E2 -2912.715} C_VEL
LIN {X 0,Y 559.151,Z 560.83,A -85,B 0,C 180,E1 -2915.323,E2 -2915.323} C_VEL
LIN {X 0,Y 559.131,Z 560.835,A -85,B 0,C 180,E1 -2918.018,E2 -2918.018} C_VEL
LIN {X 0,Y 559.171,Z 560.831,A -85,B 0,C 180,E1 -2920.811,E2 -2920.811} C_VEL
LIN {X 0,Y 559.159,Z 560.829,A -85,B 0,C 180,E1 -2923.732,E2 -2923.732} C_VEL
LIN {X 0,Y 559.142,Z 560.836,A -85,B 0,C 180,E1 -2926.804,E2 -2926.804} C_VEL
LIN {X 0,Y 559.173,Z 560.827,A -85,B 0,C 180,E1 -2929.19,E2 -2929.19} C_VEL
LIN {X 0,Y 559.131,Z 560.835,A -85,B 0,C 180,E1 -2931.983,E2 -2931.983} C_VEL
LIN {X 0,Y 559.145,Z 560.836,A -85,B 0,C 180,E1 -2934.786,E2 -2934.786} C_VEL
LIN {X 0,Y 559.172,Z 560.828,A -85,B 0,C 180,E1 -2937.362,E2 -2937.362} C_VEL
LIN {X 0,Y 559.148,Z 560.836,A -85,B 0,C 180,E1 -2940.143,E2 -2940.143} C_VEL
LIN {X 0,Y 559.17,Z 560.832,A -85,B 0,C 180,E1 -2943.098,E2 -2943.098} C_VEL
LIN {X 0,Y 559.197,Z 560.842,A -85,B 0,C 180,E1 -2944.155,E2 -2944.155} C_VEL
LIN {X 0,Y 560.678,Z 568.315,A -85,B 0,C 180,E1 -2945.171,E2 -2945.171} C_VEL
LIN {X 0,Y 560.513,Z 584.821,A -85,B 0,C 180,E1 -2947.322,E2 -2947.322} C_VEL
LIN {X 0,Y 560.054,Z 608.246,A -85,B 0,C 180,E1 -2950.374,E2 -2950.374} C_VEL
LIN {X 0,Y 559.753,Z 629.266,A -85,B 0,C 180,E1 -2953.071,E2 -2953.071} C_VEL
LIN {X 0,Y 559.51,Z 650.794,A -85,B 0,C 180,E1 -2955.799,E2 -2955.799} C_VEL
LIN {X 0,Y 560.309,Z 657.536,A -85,B 0,C 180,E1 -2955.912,E2 -2955.912} C_VEL
LIN {X 0,Y 560.063,Z 759.961,A -85,B 0,C 180,E1 -2957.246,E2 -2957.246} C_VEL
LIN {X 0,Y 559.909,Z 773.222,A -85,B 0,C 180,E1 -2957.564,E2 -2957.564} C_VEL
LIN {X 0,Y 559.771,Z 786.497,A -85,B 0,C 180,E1 -2958.045,E2 -2958.045} C_VEL
LIN {X 0,Y 559.633,Z 798.856,A -85,B 0,C 180,E1 -2958.663,E2 -2958.663} C_VEL
LIN {X 0,Y 559.439,Z 810.487,A -85,B 0,C 180,E1 -2959.413,E2 -2959.413} C_VEL
LIN {X 0,Y 559.29,Z 820.649,A -85,B 0,C 180,E1 -2960.233,E2 -2960.233} C_VEL
LIN {X 0,Y 559.134,Z 829.789,A -85,B 0,C 180,E1 -2961.143,E2 -2961.143} C_VEL
LIN {X 0,Y 559.009,Z 838.691,A -85,B 0,C 180,E1 -2962.233,E2 -2962.233} C_VEL
LIN {X 0,Y 558.925,Z 844.742,A -85,B 0,C 180,E1 -2963.14,E2 -2963.14} C_VEL
LIN {X 0,Y 558.935,Z 850.68,A -85,B 0,C 180,E1 -2964.227,E2 -2964.227} C_VEL
LIN {X 0,Y 558.827,Z 855.372,A -85,B 0,C 180,E1 -2965.311,E2 -2965.311} C_VEL
LIN {X 0,Y 558.836,Z 858.959,A -85,B 0,C 180,E1 -2966.395,E2 -2966.395} C_VEL
LIN {X 0,Y 558.799,Z 860.81,A -85,B 0,C 180,E1 -2967.116,E2 -2967.116} C_VEL
LIN {X 0,Y 558.745,Z 863.186,A -85,B 0,C 180,E1 -2968.559,E2 -2968.559} C_VEL
LIN {X 0,Y 558.74,Z 864,A -85,B 0,C 180,E1 -2970,E2 -2970} C_VEL
LIN {X 0,Y 558.745,Z 863.185,A -85,B 0,C 180,E1 -2971.441,E2 -2971.441} C_VEL
LIN {X 0,Y 558.799,Z 860.808,A -85,B 0,C 180,E1 -2972.884,E2 -2972.884} C_VEL
LIN {X 0,Y 558.844,Z 857.895,A -85,B 0,C 180,E1 -2973.966,E2 -2973.966} C_VEL
LIN {X 0,Y 558.798,Z 853.95,A -85,B 0,C 180,E1 -2975.051,E2 -2975.051} C_VEL
LIN {X 0,Y 558.921,Z 848.868,A -85,B 0,C 180,E1 -2976.135,E2 -2976.135} C_VEL
LIN {X 0,Y 558.977,Z 842.469,A -85,B 0,C 180,E1 -2977.223,E2 -2977.223} C_VEL
LIN {X 0,Y 559.099,Z 834.48,A -85,B 0,C 180,E1 -2978.311,E2 -2978.311} C_VEL
LIN {X 0,Y 559.184,Z 826.337,A -85,B 0,C 180,E1 -2979.221,E2 -2979.221} C_VEL
LIN {X 0,Y 559.355,Z 816.404,A -85,B 0,C 180,E1 -2980.131,E2 -2980.131} C_VEL
LIN {X 0,Y 559.529,Z 805.4,A -85,B 0,C 180,E1 -2980.937,E2 -2980.937} C_VEL
LIN {X 0,Y 559.671,Z 793.468,A -85,B 0,C 180,E1 -2981.627,E2 -2981.627} C_VEL
LIN {X 0,Y 559.851,Z 780.783,A -85,B 0,C 180,E1 -2982.184,E2 -2982.184} C_VEL
LIN {X 0,Y 559.972,Z 767.365,A -85,B 0,C 180,E1 -2982.595,E2 -2982.595} C_VEL
LIN {X 0,Y 560.106,Z 754.107,A -85,B 0,C 180,E1 -2982.845,E2 -2982.845} C_VEL
LIN {X 0,Y 560.181,Z 654.306,A -85,B 0,C 180,E1 -2984.133,E2 -2984.133} C_VEL
LIN {X 0,Y 559.587,Z 649.727,A -85,B 0,C 180,E1 -2984.222,E2 -2984.222} C_VEL
LIN {X 0,Y 559.907,Z 622.663,A -85,B 0,C 180,E1 -2987.212,E2 -2987.212} C_VEL
LIN {X 0,Y 560.326,Z 598.054,A -85,B 0,C 180,E1 -2989.966,E2 -2989.966} C_VEL
LIN {X 0,Y 560.782,Z 572.595,A -85,B 0,C 180,E1 -2992.861,E2 -2992.861} C_VEL
LIN {X 0,Y 560.597,Z 566.925,A -85,B 0,C 180,E1 -2993.526,E2 -2993.526} C_VEL
LIN {X 0,Y 559.204,Z 560.83,A -85,B 0,C 180,E1 -2994.304,E2 -2994.304} C_VEL
LIN {X 0,Y 559.18,Z 560.827,A -85,B 0,C 180,E1 -2996.901,E2 -2996.901} C_VEL
LIN {X 0,Y 559.149,Z 560.839,A -85,B 0,C 180,E1 -2999.857,E2 -2999.857} C_VEL
LIN {X 0,Y 559.174,Z 560.827,A -85,B 0,C 180,E1 -3002.713,E2 -3002.713} C_VEL
LIN {X 0,Y 559.156,Z 560.829,A -85,B 0,C 180,E1 -3005.321,E2 -3005.321} C_VEL
LIN {X 0,Y 559.132,Z 560.84,A -85,B 0,C 180,E1 -3008.017,E2 -3008.017} C_VEL
LIN {X 0,Y 559.174,Z 560.826,A -85,B 0,C 180,E1 -3010.81,E2 -3010.81} C_VEL
LIN {X 0,Y 559.14,Z 560.834,A -85,B 0,C 180,E1 -3013.733,E2 -3013.733} C_VEL
LIN {X 0,Y 559.163,Z 560.828,A -85,B 0,C 180,E1 -3016.8,E2 -3016.8} C_VEL
LIN {X 0,Y 559.175,Z 560.825,A -85,B 0,C 180,E1 -3019.189,E2 -3019.189} C_VEL
LIN {X 0,Y 559.131,Z 560.837,A -85,B 0,C 180,E1 -3021.982,E2 -3021.982} C_VEL
LIN {X 0,Y 559.15,Z 560.83,A -85,B 0,C 180,E1 -3024.677,E2 -3024.677} C_VEL
LIN {X 0,Y 559.167,Z 560.827,A -85,B 0,C 180,E1 -3027.361,E2 -3027.361} C_VEL
LIN {X 0,Y 559.181,Z 560.831,A -85,B 0,C 180,E1 -3030.134,E2 -3030.134} C_VEL
LIN {X 0,Y 559.175,Z 560.826,A -85,B 0,C 180,E1 -3033.169,E2 -3033.169} C_VEL
LIN {X 0,Y 559.148,Z 560.829,A -85,B 0,C 180,E1 -3035.494,E2 -3035.494} C_VEL
LIN {X 0,Y 559.168,Z 560.833,A -85,B 0,C 180,E1 -3038.624,E2 -3038.624} C_VEL
LIN {X 0,Y 559.162,Z 560.83,A -85,B 0,C 180,E1 -3040.926,E2 -3040.926} C_VEL
LIN {X 0,Y 559.161,Z 560.827,A -85,B 0,C 180,E1 -3043.948,E2 -3043.948} C_VEL
LIN {X 0,Y 559.164,Z 560.83,A -85,B 0,C 180,E1 -3046.184,E2 -3046.184} C_VEL
LIN {X 0,Y 559.201,Z 560.823,A -85,B 0,C 180,E1 -3049.134,E2 -3049.134} C_VEL
LIN {X 0,Y 559.201,Z 560.821,A -85,B 0,C 180,E1 -3052.054,E2 -3052.054} C_VEL
LIN {X 0,Y 559.255,Z 560.821,A -85,B 0,C 180,E1 -3054.953,E2 -3054.953} C_VEL
LIN {X 0,Y 559.242,Z 560.815,A -85,B 0,C 180,E1 -3057.839,E2 -3057.839} C_VEL
LIN {X 0,Y 559.27,Z 560.823,A -85,B 0,C 180,E1 -3060.72,E2 -3060.72} C_VEL
LIN {X 0,Y 559.236,Z 560.826,A -85,B 0,C 180,E1 -3062.881,E2 -3062.881} C_VEL
LIN {X 0,Y 559.227,Z 560.815,A -85,B 0,C 180,E1 -3065.77,E2 -3065.77} C_VEL
LIN {X 0,Y 559.195,Z 560.831,A -85,B 0,C 180,E1 -3068.674,E2 -3068.674} C_VEL
LIN {X 0,Y 559.199,Z 560.821,A -85,B 0,C 180,E1 -3071.601,E2 -3071.601} C_VEL
LIN {X 0,Y 559.189,Z 560.828,A -85,B 0,C 180,E1 -3074.596,E2 -3074.596} C_VEL
LIN {X 0,Y 559.154,Z 560.828,A -85,B 0,C 180,E1 -3077.557,E2 -3077.557} C_VEL
LIN {X 0,Y 559.165,Z 560.826,A -85,B 0,C 180,E1 -3079.838,E2 -3079.838} C_VEL
LIN {X 0,Y 559.133,Z 560.831,A -85,B 0,C 180,E1 -3082.153,E2 -3082.153} C_VEL
LIN {X 0,Y 559.171,Z 560.834,A -85,B 0,C 180,E1 -3085.188,E2 -3085.188} C_VEL
LIN {X 0,Y 559.187,Z 560.826,A -85,B 0,C 180,E1 -3087.712,E2 -3087.712} C_VEL
LIN {X 0,Y 559.145,Z 560.831,A -85,B 0,C 180,E1 -3090.634,E2 -3090.634} C_VEL
LIN {X 0,Y 558.482,Z 560.921,A -85,B 0,C 180,E1 -3091.235,E2 -3091.235} C_VEL
LIN {X 0,Y 555.617,Z 561.278,A -85,B 0,C 180,E1 -3092.211,E2 -3092.211} C_VEL
LIN {X 0,Y 553.203,Z 561.578,A -85,B 0,C 180,E1 -3092.997,E2 -3092.997} C_VEL
LIN {X 0,Y 552.182,Z 561.699,A -85,B 0,C 180,E1 -3093.604,E2 -3093.604} C_VEL
LIN {X 0,Y 552.108,Z 561.706,A -85,B 0,C 180,E1 -3093.809,E2 -3093.809} C_VEL
LIN {X 0,Y 552.106,Z 561.71,A -85,B 0,C 180,E1 -3096.747,E2 -3096.747} C_VEL
LIN {X 0,Y 552.129,Z 561.708,A -85,B 0,C 180,E1 -3099.527,E2 -3099.527} C_VEL
LIN {X 0,Y 552.125,Z 561.698,A -85,B 0,C 180,E1 -3102.426,E2 -3102.426} C_VEL
LIN {X 0,Y 552.093,Z 561.714,A -85,B 0,C 180,E1 -3105.564,E2 -3105.564} C_VEL
LIN {X 0,Y 552.128,Z 561.703,A -85,B 0,C 180,E1 -3108.678,E2 -3108.678} C_VEL
LIN {X 0,Y 552.116,Z 561.712,A -85,B 0,C 180,E1 -3111.412,E2 -3111.412} C_VEL
LIN {X 0,Y 552.111,Z 561.707,A -85,B 0,C 180,E1 -3114.159,E2 -3114.159} C_VEL
LIN {X 0,Y 552.122,Z 561.706,A -85,B 0,C 180,E1 -3116.816,E2 -3116.816} C_VEL
LIN {X 0,Y 552.101,Z 561.716,A -85,B 0,C 180,E1 -3119.392,E2 -3119.392} C_VEL
LIN {X 0,Y 552.106,Z 561.714,A -85,B 0,C 180,E1 -3121.902,E2 -3121.902} C_VEL
LIN {X 0,Y 552.073,Z 561.915,A -85,B 0,C 180,E1 -3123.086,E2 -3123.086} C_VEL
LIN {X 0,Y 552.055,Z 564.616,A -85,B 0,C 180,E1 -3123.694,E2 -3123.694} C_VEL
LIN {X 0,Y 553.424,Z 573.004,A -85,B 0,C 180,E1 -3123.85,E2 -3123.85} C_VEL
LIN {X 0,Y 553.086,Z 670.221,A -85,B 0,C 180,E1 -3125.133,E2 -3125.133} C_VEL
LIN {X 0,Y 552.953,Z 683.359,A -85,B 0,C 180,E1 -3125.453,E2 -3125.453} C_VEL
LIN {X 0,Y 552.849,Z 695.533,A -85,B 0,C 180,E1 -3125.897,E2 -3125.897} C_VEL
LIN {X 0,Y 552.65,Z 707.829,A -85,B 0,C 180,E1 -3126.503,E2 -3126.503} C_VEL
LIN {X 0,Y 552.446,Z 718.399,A -85,B 0,C 180,E1 -3127.17,E2 -3127.17} C_VEL
LIN {X 0,Y 552.266,Z 729.584,A -85,B 0,C 180,E1 -3128.059,E2 -3128.059} C_VEL
LIN {X 0,Y 552.107,Z 738.428,A -85,B 0,C 180,E1 -3128.925,E2 -3128.925} C_VEL
LIN {X 0,Y 551.969,Z 746.593,A -85,B 0,C 180,E1 -3129.893,E2 -3129.893} C_VEL
LIN {X 0,Y 551.868,Z 754.472,A -85,B 0,C 180,E1 -3131.051,E2 -3131.051} C_VEL
LIN {X 0,Y 551.786,Z 760.699,A -85,B 0,C 180,E1 -3132.201,E2 -3132.201} C_VEL
LIN {X 0,Y 551.749,Z 765.561,A -85,B 0,C 180,E1 -3133.346,E2 -3133.346} C_VEL
LIN {X 0,Y 551.709,Z 769.214,A -85,B 0,C 180,E1 -3134.484,E2 -3134.484} C_VEL
LIN {X 0,Y 551.687,Z 771.57,A -85,B 0,C 180,E1 -3135.506,E2 -3135.506} C_VEL
LIN {X 0,Y 551.659,Z 773.353,A -85,B 0,C 180,E1 -3136.744,E2 -3136.744} C_VEL
LIN {X 0,Y 551.658,Z 773.885,A -85,B 0,C 180,E1 -3137.492,E2 -3137.492} C_VEL
LIN {X 0,Y 551.711,Z 773.784,A -85,B 0,C 180,E1 -3138.776,E2 -3138.776} C_VEL
LIN {X 0,Y 551.677,Z 772.945,A -85,B 0,C 180,E1 -3139.727,E2 -3139.727} C_VEL
LIN {X 0,Y 551.662,Z 771.798,A -85,B 0,C 180,E1 -3140.467,E2 -3140.467} C_VEL
LIN {X 0,Y 551.686,Z 770.228,A -85,B 0,C 180,E1 -3141.207,E2 -3141.207} C_VEL
LIN {X 0,Y 551.755,Z 767.065,A -85,B 0,C 180,E1 -3142.314,E2 -3142.314} C_VEL
LIN {X 0,Y 551.823,Z 762.846,A -85,B 0,C 180,E1 -3143.418,E2 -3143.418} C_VEL
LIN {X 0,Y 551.8,Z 756.47,A -85,B 0,C 180,E1 -3144.702,E2 -3144.702} C_VEL
LIN {X 0,Y 551.944,Z 749.484,A -85,B 0,C 180,E1 -3145.801,E2 -3145.801} C_VEL
LIN {X 0,Y 552.034,Z 740.848,A -85,B 0,C 180,E1 -3146.898,E2 -3146.898} C_VEL
LIN {X 0,Y 552.242,Z 731.004,A -85,B 0,C 180,E1 -3147.903,E2 -3147.903} C_VEL
LIN {X 0,Y 552.383,Z 719.857,A -85,B 0,C 180,E1 -3148.815,E2 -3148.815} C_VEL
LIN {X 0,Y 552.57,Z 708.615,A -85,B 0,C 180,E1 -3149.545,E2 -3149.545} C_VEL
LIN {X 0,Y 552.805,Z 695.793,A -85,B 0,C 180,E1 -3150.182,E2 -3150.182} C_VEL
LIN {X 0,Y 553.003,Z 683.328,A -85,B 0,C 180,E1 -3150.637,E2 -3150.637} C_VEL
LIN {X 0,Y 553.111,Z 670.249,A -85,B 0,C 180,E1 -3150.956,E2 -3150.956} C_VEL
LIN {X 0,Y 553.302,Z 570.595,A -85,B 0,C 180,E1 -3152.275,E2 -3152.275} C_VEL
LIN {X 0,Y 552.193,Z 563.665,A -85,B 0,C 180,E1 -3152.416,E2 -3152.416} C_VEL
LIN {X 0,Y 552.206,Z 561.699,A -85,B 0,C 180,E1 -3152.827,E2 -3152.827} C_VEL
LIN {X 0,Y 552.198,Z 561.703,A -85,B 0,C 180,E1 -3155.844,E2 -3155.844} C_VEL
LIN {X 0,Y 552.145,Z 561.703,A -85,B 0,C 180,E1 -3158.786,E2 -3158.786} C_VEL
LIN {X 0,Y 552.166,Z 561.704,A -85,B 0,C 180,E1 -3161.75,E2 -3161.75} C_VEL
LIN {X 0,Y 552.139,Z 561.704,A -85,B 0,C 180,E1 -3164.748,E2 -3164.748} C_VEL
LIN {X 0,Y 552.113,Z 561.712,A -85,B 0,C 180,E1 -3167.788,E2 -3167.788} C_VEL
LIN {X 0,Y 552.131,Z 561.712,A -85,B 0,C 180,E1 -3170.101,E2 -3170.101} C_VEL
LIN {X 0,Y 552.094,Z 561.712,A -85,B 0,C 180,E1 -3172.45,E2 -3172.45} C_VEL
LIN {X 0,Y 552.156,Z 561.702,A -85,B 0,C 180,E1 -3175.35,E2 -3175.35} C_VEL
LIN {X 0,Y 552.126,Z 561.713,A -85,B 0,C 180,E1 -3178.097,E2 -3178.097} C_VEL
LIN {X 0,Y 552.159,Z 561.705,A -85,B 0,C 180,E1 -3181.243,E2 -3181.243} C_VEL
LIN {X 0,Y 552.158,Z 563.847,A -85,B 0,C 180,E1 -3181.696,E2 -3181.696} C_VEL
LIN {X 0,Y 553.432,Z 572.399,A -85,B 0,C 180,E1 -3181.842,E2 -3181.842} C_VEL
LIN {X 0,Y 553.107,Z 669.035,A -85,B 0,C 180,E1 -3183.118,E2 -3183.118} C_VEL
LIN {X 0,Y 553.029,Z 680.174,A -85,B 0,C 180,E1 -3183.368,E2 -3183.368} C_VEL
LIN {X 0,Y 552.918,Z 689.778,A -85,B 0,C 180,E1 -3183.676,E2 -3183.676} C_VEL
LIN {X 0,Y 552.747,Z 699.923,A -85,B 0,C 180,E1 -3184.1,E2 -3184.1} C_VEL
LIN {X 0,Y 552.632,Z 710.055,A -85,B 0,C 180,E1 -3184.639,E2 -3184.639} C_VEL
LIN {X 0,Y 552.407,Z 720.413,A -85,B 0,C 180,E1 -3185.32,E2 -3185.32} C_VEL
LIN {X 0,Y 552.262,Z 730.808,A -85,B 0,C 180,E1 -3186.167,E2 -3186.167} C_VEL
LIN {X 0,Y 552.066,Z 740.926,A -85,B 0,C 180,E1 -3187.206,E2 -3187.206} C_VEL
LIN {X 0,Y 551.925,Z 748.876,A -85,B 0,C 180,E1 -3188.211,E2 -3188.211} C_VEL
LIN {X 0,Y 551.868,Z 755.687,A -85,B 0,C 180,E1 -3189.264,E2 -3189.264} C_VEL
LIN {X 0,Y 551.769,Z 762.145,A -85,B 0,C 180,E1 -3190.51,E2 -3190.51} C_VEL
LIN {X 0,Y 551.749,Z 767.524,A -85,B 0,C 180,E1 -3191.919,E2 -3191.919} C_VEL
LIN {X 0,Y 551.674,Z 770.393,A -85,B 0,C 180,E1 -3192.949,E2 -3192.949} C_VEL
LIN {X 0,Y 551.664,Z 773.042,A -85,B 0,C 180,E1 -3194.486,E2 -3194.486} C_VEL
LIN {X 0,Y 551.664,Z 773.838,A -85,B 0,C 180,E1 -3195.518,E2 -3195.518} C_VEL
LIN {X 0,Y 551.663,Z 773.841,A -85,B 0,C 180,E1 -3196.564,E2 -3196.564} C_VEL
LIN {X 0,Y 551.652,Z 773.001,A -85,B 0,C 180,E1 -3197.637,E2 -3197.637} C_VEL
LIN {X 0,Y 551.682,Z 771.252,A -85,B 0,C 180,E1 -3198.729,E2 -3198.729} C_VEL
LIN {X 0,Y 551.707,Z 768.488,A -85,B 0,C 180,E1 -3199.845,E2 -3199.845} C_VEL
LIN {X 0,Y 551.754,Z 764.589,A -85,B 0,C 180,E1 -3200.984,E2 -3200.984} C_VEL
LIN {X 0,Y 551.79,Z 759.367,A -85,B 0,C 180,E1 -3202.153,E2 -3202.153} C_VEL
LIN {X 0,Y 551.88,Z 752.569,A -85,B 0,C 180,E1 -3203.347,E2 -3203.347} C_VEL
LIN {X 0,Y 552.012,Z 745.099,A -85,B 0,C 180,E1 -3204.388,E2 -3204.388} C_VEL
LIN {X 0,Y 552.177,Z 736.498,A -85,B 0,C 180,E1 -3205.364,E2 -3205.364} C_VEL
LIN {X 0,Y 552.284,Z 727.931,A -85,B 0,C 180,E1 -3206.17,E2 -3206.17} C_VEL
LIN {X 0,Y 552.44,Z 719.469,A -85,B 0,C 180,E1 -3206.836,E2 -3206.836} C_VEL
LIN {X 0,Y 552.591,Z 710.798,A -85,B 0,C 180,E1 -3207.408,E2 -3207.408} C_VEL
LIN {X 0,Y 552.72,Z 701.324,A -85,B 0,C 180,E1 -3207.924,E2 -3207.924} C_VEL
LIN {X 0,Y 552.871,Z 691.361,A -85,B 0,C 180,E1 -3208.357,E2 -3208.357} C_VEL
LIN {X 0,Y 552.984,Z 680.469,A -85,B 0,C 180,E1 -3208.715,E2 -3208.715} C_VEL
LIN {X 0,Y 553.072,Z 669.776,A -85,B 0,C 180,E1 -3208.96,E2 -3208.96} C_VEL
LIN {X 0,Y 553.398,Z 578.554,A -85,B 0,C 180,E1 -3210.168,E2 -3210.168} C_VEL
LIN {X 0,Y 553.177,Z 571.057,A -85,B 0,C 180,E1 -3210.272,E2 -3210.272} C_VEL
LIN {X 0,Y 552.077,Z 564.64,A -85,B 0,C 180,E1 -3210.39,E2 -3210.39} C_VEL
LIN {X 0,Y 552.097,Z 561.715,A -85,B 0,C 180,E1 -3211.071,E2 -3211.071} C_VEL
LIN {X 0,Y 552.127,Z 561.706,A -85,B 0,C 180,E1 -3213.544,E2 -3213.544} C_VEL
LIN {X 0,Y 552.103,Z 561.716,A -85,B 0,C 180,E1 -3216.42,E2 -3216.42} C_VEL
LIN {X 0,Y 552.118,Z 561.708,A -85,B 0,C 180,E1 -3219.12,E2 -3219.12} C_VEL
LIN {X 0,Y 552.123,Z 561.705,A -85,B 0,C 180,E1 -3221.444,E2 -3221.444} C_VEL
LIN {X 0,Y 552.112,Z 561.707,A -85,B 0,C 180,E1 -3223.737,E2 -3223.737} C_VEL
LIN {X 0,Y 552.128,Z 561.707,A -85,B 0,C 180,E1 -3226.004,E2 -3226.004} C_VEL
LIN {X 0,Y 552.169,Z 561.702,A -85,B 0,C 180,E1 -3228.993,E2 -3228.993} C_VEL
LIN {X 0,Y 552.157,Z 561.703,A -85,B 0,C 180,E1 -3231.952,E2 -3231.952} C_VEL
LIN {X 0,Y 552.227,Z 561.696,A -85,B 0,C 180,E1 -3234.889,E2 -3234.889} C_VEL
LIN {X 0,Y 552.214,Z 561.693,A -85,B 0,C 180,E1 -3237.812,E2 -3237.812} C_VEL
LIN {X 0,Y 552.237,Z 561.697,A -85,B 0,C 180,E1 -3240.729,E2 -3240.729} C_VEL
LIN {X 0,Y 552.202,Z 561.698,A -85,B 0,C 180,E1 -3242.918,E2 -3242.918} C_VEL
LIN {X 0,Y 552.198,Z 561.696,A -85,B 0,C 180,E1 -3245.844,E2 -3245.844} C_VEL
LIN {X 0,Y 552.163,Z 561.704,A -85,B 0,C 180,E1 -3248.786,E2 -3248.786} C_VEL
LIN {X 0,Y 552.155,Z 561.7,A -85,B 0,C 180,E1 -3251.751,E2 -3251.751} C_VEL
LIN {X 0,Y 552.126,Z 561.709,A -85,B 0,C 180,E1 -3254.749,E2 -3254.749} C_VEL
LIN {X 0,Y 552.107,Z 561.706,A -85,B 0,C 180,E1 -3257.789,E2 -3257.789} C_VEL
LIN {X 0,Y 552.126,Z 561.707,A -85,B 0,C 180,E1 -3260.101,E2 -3260.101} C_VEL
LIN {X 0,Y 552.106,Z 561.715,A -85,B 0,C 180,E1 -3262.45,E2 -3262.45} C_VEL
LIN {X 0,Y 552.148,Z 561.702,A -85,B 0,C 180,E1 -3265.351,E2 -3265.351} C_VEL
LIN {X 0,Y 552.12,Z 561.707,A -85,B 0,C 180,E1 -3268.098,E2 -3268.098} C_VEL
LIN {X 0,Y 552.107,Z 561.715,A -85,B 0,C 180,E1 -3270.609,E2 -3270.609} C_VEL
LIN {X 0,Y 552.122,Z 561.705,A -85,B 0,C 180,E1 -3273.186,E2 -3273.186} C_VEL
LIN {X 0,Y 552.107,Z 561.708,A -85,B 0,C 180,E1 -3275.842,E2 -3275.842} C_VEL
LIN {X 0,Y 552.121,Z 561.706,A -85,B 0,C 180,E1 -3279.063,E2 -3279.063} C_VEL
LIN {X 0,Y 552.135,Z 561.703,A -85,B 0,C 180,E1 -3281.445,E2 -3281.445} C_VEL
LIN {X 0,Y 552.092,Z 561.719,A -85,B 0,C 180,E1 -3284.533,E2 -3284.533} C_VEL
LIN {X 0,Y 552.127,Z 561.705,A -85,B 0,C 180,E1 -3287.585,E2 -3287.585} C_VEL
LIN {X 0,Y 552.146,Z 561.712,A -85,B 0,C 180,E1 -3290.475,E2 -3290.475} C_VEL
LIN {X 0,Y 552.107,Z 561.707,A -85,B 0,C 180,E1 -3293.317,E2 -3293.317} C_VEL
LIN {X 0,Y 552.128,Z 561.707,A -85,B 0,C 180,E1 -3295.94,E2 -3295.94} C_VEL
LIN {X 0,Y 552.118,Z 561.714,A -85,B 0,C 180,E1 -3298.541,E2 -3298.541} C_VEL
LIN {X 0,Y 552.124,Z 561.707,A -85,B 0,C 180,E1 -3301.439,E2 -3301.439} C_VEL
LIN {X 0,Y 552.156,Z 561.725,A -85,B 0,C 180,E1 -3304.003,E2 -3304.003} C_VEL
LIN {X 0,Y 553.667,Z 569.223,A -85,B 0,C 180,E1 -3305.042,E2 -3305.042} C_VEL
LIN {X 0,Y 553.666,Z 584.559,A -85,B 0,C 180,E1 -3307.026,E2 -3307.026} C_VEL
LIN {X 0,Y 553.183,Z 607.916,A -85,B 0,C 180,E1 -3310.076,E2 -3310.076} C_VEL
LIN {X 0,Y 552.774,Z 630.396,A -85,B 0,C 180,E1 -3312.997,E2 -3312.997} C_VEL
LIN {X 0,Y 552.53,Z 650.794,A -85,B 0,C 180,E1 -3315.616,E2 -3315.616} C_VEL
LIN {X 0,Y 553.434,Z 658.156,A -85,B 0,C 180,E1 -3315.742,E2 -3315.742} C_VEL
LIN {X 0,Y 553.165,Z 759.961,A -85,B 0,C 180,E1 -3317.084,E2 -3317.084} C_VEL
LIN {X 0,Y 553.012,Z 772.46,A -85,B 0,C 180,E1 -3317.384,E2 -3317.384} C_VEL
LIN {X 0,Y 552.859,Z 785.37,A -85,B 0,C 180,E1 -3317.846,E2 -3317.846} C_VEL
LIN {X 0,Y 552.689,Z 797.677,A -85,B 0,C 180,E1 -3318.45,E2 -3318.45} C_VEL
LIN {X 0,Y 552.478,Z 809.203,A -85,B 0,C 180,E1 -3319.186,E2 -3319.186} C_VEL
LIN {X 0,Y 552.269,Z 819.605,A -85,B 0,C 180,E1 -3320.015,E2 -3320.015} C_VEL
LIN {X 0,Y 552.125,Z 828.115,A -85,B 0,C 180,E1 -3320.845,E2 -3320.845} C_VEL
LIN {X 0,Y 552.013,Z 835.962,A -85,B 0,C 180,E1 -3321.765,E2 -3321.765} C_VEL
LIN {X 0,Y 551.889,Z 843.623,A -85,B 0,C 180,E1 -3322.868,E2 -3322.868} C_VEL
LIN {X 0,Y 551.867,Z 850.68,A -85,B 0,C 180,E1 -3324.153,E2 -3324.153} C_VEL
LIN {X 0,Y 551.725,Z 855.372,A -85,B 0,C 180,E1 -3325.251,E2 -3325.251} C_VEL
LIN {X 0,Y 551.751,Z 858.96,A -85,B 0,C 180,E1 -3326.349,E2 -3326.349} C_VEL
LIN {X 0,Y 551.724,Z 860.81,A -85,B 0,C 180,E1 -3327.079,E2 -3327.079} C_VEL
LIN {X 0,Y 551.645,Z 863.186,A -85,B 0,C 180,E1 -3328.54,E2 -3328.54} C_VEL
LIN {X 0,Y 551.64,Z 864,A -85,B 0,C 180,E1 -3330,E2 -3330} C_VEL
LIN {X 0,Y 551.645,Z 863.185,A -85,B 0,C 180,E1 -3331.46,E2 -3331.46} C_VEL
LIN {X 0,Y 551.724,Z 860.808,A -85,B 0,C 180,E1 -3332.921,E2 -3332.921} C_VEL
LIN {X 0,Y 551.764,Z 857.895,A -85,B 0,C 180,E1 -3334.017,E2 -3334.017} C_VEL
LIN {X 0,Y 551.724,Z 853.95,A -85,B 0,C 180,E1 -3335.116,E2 -3335.116} C_VEL
LIN {X 0,Y 551.803,Z 848.19,A -85,B 0,C 180,E1 -3336.341,E2 -3336.341} C_VEL
LIN {X 0,Y 551.926,Z 841.238,A -85,B 0,C 180,E1 -3337.499,E2 -3337.499} C_VEL
LIN {X 0,Y 552.082,Z 832.993,A -85,B 0,C 180,E1 -3338.602,E2 -3338.602} C_VEL
LIN {X 0,Y 552.221,Z 824.541,A -85,B 0,C 180,E1 -3339.523,E2 -3339.523} C_VEL
LIN {X 0,Y 552.425,Z 814.1,A -85,B 0,C 180,E1 -3340.445,E2 -3340.445} C_VEL
LIN {X 0,Y 552.599,Z 803.292,A -85,B 0,C 180,E1 -3341.213,E2 -3341.213} C_VEL
LIN {X 0,Y 552.781,Z 792.415,A -85,B 0,C 180,E1 -3341.83,E2 -3341.83} C_VEL
LIN {X 0,Y 552.932,Z 780.78,A -85,B 0,C 180,E1 -3342.339,E2 -3342.339} C_VEL
LIN {X 0,Y 553.028,Z 767.365,A -85,B 0,C 180,E1 -3342.756,E2 -3342.756} C_VEL
LIN {X 0,Y 553.184,Z 754.107,A -85,B 0,C 180,E1 -3343.009,E2 -3343.009} C_VEL
LIN {X 0,Y 553.412,Z 655.747,A -85,B 0,C 180,E1 -3344.29,E2 -3344.29} C_VEL
LIN {X 0,Y 552.613,Z 649.727,A -85,B 0,C 180,E1 -3344.406,E2 -3344.406} C_VEL
LIN {X 0,Y 552.98,Z 624.081,A -85,B 0,C 180,E1 -3347.275,E2 -3347.275} C_VEL
LIN {X 0,Y 553.47,Z 597.884,A -85,B 0,C 180,E1 -3350.244,E2 -3350.244} C_VEL
LIN {X 0,Y 553.91,Z 574.063,A -85,B 0,C 180,E1 -3352.964,E2 -3352.964} C_VEL
LIN {X 0,Y 553.884,Z 569.396,A -85,B 0,C 180,E1 -3353.495,E2 -3353.495} C_VEL
LIN {X 0,Y 552.16,Z 561.706,A -85,B 0,C 180,E1 -3354.46,E2 -3354.46} C_VEL
LIN {X 0,Y 552.149,Z 561.705,A -85,B 0,C 180,E1 -3357.272,E2 -3357.272} C_VEL
LIN {X 0,Y 552.117,Z 561.714,A -85,B 0,C 180,E1 -3360.05,E2 -3360.05} C_VEL
LIN {X 0,Y 552.129,Z 561.704,A -85,B 0,C 180,E1 -3362.848,E2 -3362.848} C_VEL
LIN {X 0,Y 552.106,Z 561.709,A -85,B 0,C 180,E1 -3365.444,E2 -3365.444} C_VEL
LIN {X 0,Y 552.095,Z 561.716,A -85,B 0,C 180,E1 -3367.885,E2 -3367.885} C_VEL
LIN {X 0,Y 552.14,Z 561.706,A -85,B 0,C 180,E1 -3370.477,E2 -3370.477} C_VEL
LIN {X 0,Y 552.114,Z 561.707,A -85,B 0,C 180,E1 -3373.484,E2 -3373.484} C_VEL
LIN {X 0,Y 552.115,Z 561.709,A -85,B 0,C 180,E1 -3376.577,E2 -3376.577} C_VEL
LIN {X 0,Y 552.139,Z 561.703,A -85,B 0,C 180,E1 -3379.521,E2 -3379.521} C_VEL
LIN {X 0,Y 552.09,Z 561.717,A -85,B 0,C 180,E1 -3382.336,E2 -3382.336} C_VEL
LIN {X 0,Y 552.121,Z 561.702,A -85,B 0,C 180,E1 -3385.054,E2 -3385.054} C_VEL
LIN {X 0,Y 552.12,Z 561.706,A -85,B 0,C 180,E1 -3387.682,E2 -3387.682} C_VEL
LIN {X 0,Y 552.137,Z 561.711,A -85,B 0,C 180,E1 -3390.236,E2 -3390.236} C_VEL
LIN {X 0,Y 552.14,Z 561.704,A -85,B 0,C 180,E1 -3392.997,E2 -3392.997} C_VEL
LIN {X 0,Y 552.105,Z 561.707,A -85,B 0,C 180,E1 -3395.161,E2 -3395.161} C_VEL
LIN {X 0,Y 552.087,Z 561.705,A -85,B 0,C 180,E1 -3397.549,E2 -3397.549} C_VEL
LIN {X 0,Y 552.14,Z 561.711,A -85,B 0,C 180,E1 -3400.373,E2 -3400.373} C_VEL
LIN {X 0,Y 552.147,Z 561.701,A -85,B 0,C 180,E1 -3402.977,E2 -3402.977} C_VEL
LIN {X 0,Y 552.127,Z 561.705,A -85,B 0,C 180,E1 -3406.004,E2 -3406.004} C_VEL
LIN {X 0,Y 552.169,Z 561.701,A -85,B 0,C 180,E1 -3408.993,E2 -3408.993} C_VEL
LIN {X 0,Y 552.155,Z 561.698,A -85,B 0,C 180,E1 -3411.951,E2 -3411.951} C_VEL
LIN {X 0,Y 552.229,Z 561.697,A -85,B 0,C 180,E1 -3414.889,E2 -3414.889} C_VEL
LIN {X 0,Y 552.214,Z 561.69,A -85,B 0,C 180,E1 -3417.812,E2 -3417.812} C_VEL
LIN {X 0,Y 552.239,Z 561.699,A -85,B 0,C 180,E1 -3420.729,E2 -3420.729} C_VEL
LIN {X 0,Y 552.202,Z 561.701,A -85,B 0,C 180,E1 -3422.918,E2 -3422.918} C_VEL
LIN {X 0,Y 552.198,Z 561.691,A -85,B 0,C 180,E1 -3425.844,E2 -3425.844} C_VEL
LIN {X 0,Y 552.162,Z 561.709,A -85,B 0,C 180,E1 -3428.786,E2 -3428.786} C_VEL
LIN {X 0,Y 552.154,Z 561.698,A -85,B 0,C 180,E1 -3431.751,E2 -3431.751} C_VEL
LIN {X 0,Y 552.126,Z 561.71,A -85,B 0,C 180,E1 -3434.749,E2 -3434.749} C_VEL
LIN {X 0,Y 552.105,Z 561.705,A -85,B 0,C 180,E1 -3437.789,E2 -3437.789} C_VEL
LIN {X 0,Y 552.124,Z 561.703,A -85,B 0,C 180,E1 -3440.102,E2 -3440.102} C_VEL
LIN {X 0,Y 552.087,Z 561.711,A -85,B 0,C 180,E1 -3442.451,E2 -3442.451} C_VEL
LIN {X 0,Y 552.148,Z 561.706,A -85,B 0,C 180,E1 -3445.351,E2 -3445.351} C_VEL
LIN {X 0,Y 552.119,Z 561.705,A -85,B 0,C 180,E1 -3448.098,E2 -3448.098} C_VEL
LIN {X 0,Y 552.105,Z 561.707,A -85,B 0,C 180,E1 -3450.629,E2 -3450.629} C_VEL
LIN {X 0,Y 552.115,Z 561.713,A -85,B 0,C 180,E1 -3453.186,E2 -3453.186} C_VEL
LIN {X 0,Y 552.108,Z 561.706,A -85,B 0,C 180,E1 -3453.809,E2 -3453.809} C_VEL
LIN {X 0,Y 551.466,Z 561.786,A -85,B 0,C 180,E1 -3454.418,E2 -3454.418} C_VEL
LIN {X 0,Y 548.622,Z 562.147,A -85,B 0,C 180,E1 -3455.406,E2 -3455.406} C_VEL
LIN {X 0,Y 546.2,Z 562.448,A -85,B 0,C 180,E1 -3456.201,E2 -3456.201} C_VEL
LIN {X 0,Y 545.153,Z 562.578,A -85,B 0,C 180,E1 -3456.815,E2 -3456.815} C_VEL
LIN {X 0,Y 545.065,Z 562.59,A -85,B 0,C 180,E1 -3457.023,E2 -3457.023} C_VEL
LIN {X 0,Y 545.069,Z 562.582,A -85,B 0,C 180,E1 -3460.143,E2 -3460.143} C_VEL
LIN {X 0,Y 545.082,Z 562.582,A -85,B 0,C 180,E1 -3463.107,E2 -3463.107} C_VEL
LIN {X 0,Y 545.045,Z 562.586,A -85,B 0,C 180,E1 -3466.227,E2 -3466.227} C_VEL
LIN {X 0,Y 545.091,Z 562.581,A -85,B 0,C 180,E1 -3468.888,E2 -3468.888} C_VEL
LIN {X 0,Y 545.05,Z 562.588,A -85,B 0,C 180,E1 -3471.764,E2 -3471.764} C_VEL
LIN {X 0,Y 545.063,Z 562.584,A -85,B 0,C 180,E1 -3474.535,E2 -3474.535} C_VEL
LIN {X 0,Y 545.08,Z 562.589,A -85,B 0,C 180,E1 -3477.213,E2 -3477.213} C_VEL
LIN {X 0,Y 545.063,Z 562.59,A -85,B 0,C 180,E1 -3479.811,E2 -3479.811} C_VEL
LIN {X 0,Y 545.088,Z 562.585,A -85,B 0,C 180,E1 -3482.345,E2 -3482.345} C_VEL
LIN {X 0,Y 545.015,Z 562.778,A -85,B 0,C 180,E1 -3483.085,E2 -3483.085} C_VEL
LIN {X 0,Y 544.996,Z 564.656,A -85,B 0,C 180,E1 -3483.513,E2 -3483.513} C_VEL
LIN {X 0,Y 546.555,Z 573.781,A -85,B 0,C 180,E1 -3483.678,E2 -3483.678} C_VEL
LIN {X 0,Y 546.188,Z 670.646,A -85,B 0,C 180,E1 -3484.976,E2 -3484.976} C_VEL
LIN {X 0,Y 546.007,Z 683.599,A -85,B 0,C 180,E1 -3485.297,E2 -3485.297} C_VEL
LIN {X 0,Y 545.885,Z 695.51,A -85,B 0,C 180,E1 -3485.739,E2 -3485.739} C_VEL
LIN {X 0,Y 545.681,Z 708.021,A -85,B 0,C 180,E1 -3486.365,E2 -3486.365} C_VEL
LIN {X 0,Y 545.447,Z 718.839,A -85,B 0,C 180,E1 -3487.061,E2 -3487.061} C_VEL
LIN {X 0,Y 545.235,Z 729.815,A -85,B 0,C 180,E1 -3487.951,E2 -3487.951} C_VEL
LIN {X 0,Y 545.059,Z 738.715,A -85,B 0,C 180,E1 -3488.837,E2 -3488.837} C_VEL
LIN {X 0,Y 544.908,Z 746.978,A -85,B 0,C 180,E1 -3489.838,E2 -3489.838} C_VEL
LIN {X 0,Y 544.791,Z 754.651,A -85,B 0,C 180,E1 -3490.99,E2 -3490.99} C_VEL
LIN {X 0,Y 544.722,Z 760.94,A -85,B 0,C 180,E1 -3492.176,E2 -3492.176} C_VEL
LIN {X 0,Y 544.653,Z 766.366,A -85,B 0,C 180,E1 -3493.509,E2 -3493.509} C_VEL
LIN {X 0,Y 544.633,Z 768.763,A -85,B 0,C 180,E1 -3494.277,E2 -3494.277} C_VEL
LIN {X 0,Y 544.588,Z 771.508,A -85,B 0,C 180,E1 -3495.441,E2 -3495.441} C_VEL
LIN {X 0,Y 544.558,Z 773.184,A -85,B 0,C 180,E1 -3496.567,E2 -3496.567} C_VEL
LIN {X 0,Y 544.569,Z 773.798,A -85,B 0,C 180,E1 -3497.327,E2 -3497.327} C_VEL
LIN {X 0,Y 544.621,Z 773.815,A -85,B 0,C 180,E1 -3498.736,E2 -3498.736} C_VEL
LIN {X 0,Y 544.58,Z 773.112,A -85,B 0,C 180,E1 -3499.591,E2 -3499.591} C_VEL
LIN {X 0,Y 544.584,Z 772.082,A -85,B 0,C 180,E1 -3500.342,E2 -3500.342} C_VEL
LIN {X 0,Y 544.578,Z 770.599,A -85,B 0,C 180,E1 -3501.091,E2 -3501.091} C_VEL
LIN {X 0,Y 544.66,Z 767.576,A -85,B 0,C 180,E1 -3502.213,E2 -3502.213} C_VEL
LIN {X 0,Y 544.735,Z 763.09,A -85,B 0,C 180,E1 -3503.43,E2 -3503.43} C_VEL
LIN {X 0,Y 544.747,Z 758.296,A -85,B 0,C 180,E1 -3504.447,E2 -3504.447} C_VEL
LIN {X 0,Y 544.844,Z 751.777,A -85,B 0,C 180,E1 -3505.561,E2 -3505.561} C_VEL
LIN {X 0,Y 544.959,Z 743.708,A -85,B 0,C 180,E1 -3506.673,E2 -3506.673} C_VEL
LIN {X 0,Y 545.123,Z 735.461,A -85,B 0,C 180,E1 -3507.599,E2 -3507.599} C_VEL
LIN {X 0,Y 545.291,Z 725.379,A -85,B 0,C 180,E1 -3508.523,E2 -3508.523} C_VEL
LIN {X 0,Y 545.477,Z 714.127,A -85,B 0,C 180,E1 -3509.354,E2 -3509.354} C_VEL
LIN {X 0,Y 545.778,Z 702.949,A -85,B 0,C 180,E1 -3510,E2 -3510} C_VEL
LIN {X 0,Y 545.945,Z 690.503,A -85,B 0,C 180,E1 -3510.553,E2 -3510.553} C_VEL
LIN {X 0,Y 546.126,Z 677.326,A -85,B 0,C 180,E1 -3510.968,E2 -3510.968} C_VEL
LIN {X 0,Y 546.24,Z 664.199,A -85,B 0,C 180,E1 -3511.221,E2 -3511.221} C_VEL
LIN {X 0,Y 546.431,Z 571.475,A -85,B 0,C 180,E1 -3512.446,E2 -3512.446} C_VEL
LIN {X 0,Y 545.174,Z 563.763,A -85,B 0,C 180,E1 -3512.586,E2 -3512.586} C_VEL
LIN {X 0,Y 545.183,Z 562.574,A -85,B 0,C 180,E1 -3512.863,E2 -3512.863} C_VEL
LIN {X 0,Y 545.17,Z 562.58,A -85,B 0,C 180,E1 -3515.919,E2 -3515.919} C_VEL
LIN {X 0,Y 545.105,Z 562.58,A -85,B 0,C 180,E1 -3518.9,E2 -3518.9} C_VEL
LIN {X 0,Y 545.138,Z 562.582,A -85,B 0,C 180,E1 -3521.904,E2 -3521.904} C_VEL
LIN {X 0,Y 545.088,Z 562.581,A -85,B 0,C 180,E1 -3524.943,E2 -3524.943} C_VEL
LIN {X 0,Y 545.081,Z 562.591,A -85,B 0,C 180,E1 -3528.025,E2 -3528.025} C_VEL
LIN {X 0,Y 545.096,Z 562.584,A -85,B 0,C 180,E1 -3530.371,E2 -3530.371} C_VEL
LIN {X 0,Y 545.08,Z 562.585,A -85,B 0,C 180,E1 -3533.559,E2 -3533.559} C_VEL
LIN {X 0,Y 545.08,Z 562.592,A -85,B 0,C 180,E1 -3536,E2 -3536} C_VEL
LIN {X 0,Y 545.09,Z 562.584,A -85,B 0,C 180,E1 -3538.748,E2 -3538.748} C_VEL
LIN {X 0,Y 545.106,Z 562.75,A -85,B 0,C 180,E1 -3541.301,E2 -3541.301} C_VEL
LIN {X 0,Y 545.116,Z 563.726,A -85,B 0,C 180,E1 -3541.495,E2 -3541.495} C_VEL
LIN {X 0,Y 546.549,Z 573.2,A -85,B 0,C 180,E1 -3541.67,E2 -3541.67} C_VEL
LIN {X 0,Y 546.205,Z 668.618,A -85,B 0,C 180,E1 -3542.945,E2 -3542.945} C_VEL
LIN {X 0,Y 546.096,Z 679.389,A -85,B 0,C 180,E1 -3543.183,E2 -3543.183} C_VEL
LIN {X 0,Y 545.957,Z 689.208,A -85,B 0,C 180,E1 -3543.495,E2 -3543.495} C_VEL
LIN {X 0,Y 545.822,Z 698.84,A -85,B 0,C 180,E1 -3543.895,E2 -3543.895} C_VEL
LIN {X 0,Y 545.681,Z 708.684,A -85,B 0,C 180,E1 -3544.411,E2 -3544.411} C_VEL
LIN {X 0,Y 545.508,Z 717.579,A -85,B 0,C 180,E1 -3544.98,E2 -3544.98} C_VEL
LIN {X 0,Y 545.326,Z 725.438,A -85,B 0,C 180,E1 -3545.577,E2 -3545.577} C_VEL
LIN {X 0,Y 545.156,Z 734.175,A -85,B 0,C 180,E1 -3546.371,E2 -3546.371} C_VEL
LIN {X 0,Y 545.042,Z 740.857,A -85,B 0,C 180,E1 -3547.084,E2 -3547.084} C_VEL
LIN {X 0,Y 544.87,Z 748.884,A -85,B 0,C 180,E1 -3548.112,E2 -3548.112} C_VEL
LIN {X 0,Y 544.818,Z 754.448,A -85,B 0,C 180,E1 -3548.965,E2 -3548.965} C_VEL
LIN {X 0,Y 544.752,Z 759.726,A -85,B 0,C 180,E1 -3549.934,E2 -3549.934} C_VEL
LIN {X 0,Y 544.679,Z 763.508,A -85,B 0,C 180,E1 -3550.76,E2 -3550.76} C_VEL
LIN {X 0,Y 544.663,Z 766.506,A -85,B 0,C 180,E1 -3551.548,E2 -3551.548} C_VEL
LIN {X 0,Y 544.598,Z 769.766,A -85,B 0,C 180,E1 -3552.643,E2 -3552.643} C_VEL
LIN {X 0,Y 544.565,Z 772.035,A -85,B 0,C 180,E1 -3553.72,E2 -3553.72} C_VEL
LIN {X 0,Y 544.552,Z 773.713,A -85,B 0,C 180,E1 -3555.22,E2 -3555.22} C_VEL
LIN {X 0,Y 544.563,Z 773.953,A -85,B 0,C 180,E1 -3556.278,E2 -3556.278} C_VEL
LIN {X 0,Y 544.542,Z 773.352,A -85,B 0,C 180,E1 -3557.361,E2 -3557.361} C_VEL
LIN {X 0,Y 544.579,Z 771.09,A -85,B 0,C 180,E1 -3558.839,E2 -3558.839} C_VEL
LIN {X 0,Y 544.631,Z 768.702,A -85,B 0,C 180,E1 -3559.819,E2 -3559.819} C_VEL
LIN {X 0,Y 544.661,Z 765.601,A -85,B 0,C 180,E1 -3560.782,E2 -3560.782} C_VEL
LIN {X 0,Y 544.691,Z 760.906,A -85,B 0,C 180,E1 -3561.91,E2 -3561.91} C_VEL
LIN {X 0,Y 544.763,Z 755.64,A -85,B 0,C 180,E1 -3562.922,E2 -3562.922} C_VEL
LIN {X 0,Y 544.878,Z 748.731,A -85,B 0,C 180,E1 -3564,E2 -3564} C_VEL
LIN {X 0,Y 545.033,Z 741.048,A -85,B 0,C 180,E1 -3564.983,E2 -3564.983} C_VEL
LIN {X 0,Y 545.232,Z 731.291,A -85,B 0,C 180,E1 -3566.006,E2 -3566.006} C_VEL
LIN {X 0,Y 545.435,Z 720.823,A -85,B 0,C 180,E1 -3566.878,E2 -3566.878} C_VEL
LIN {X 0,Y 545.63,Z 710.406,A -85,B 0,C 180,E1 -3567.578,E2 -3567.578} C_VEL
LIN {X 0,Y 545.758,Z 701.331,A -85,B 0,C 180,E1 -3568.077,E2 -3568.077} C_VEL
LIN {X 0,Y 545.913,Z 691.233,A -85,B 0,C 180,E1 -3568.52,E2 -3568.52} C_VEL
LIN {X 0,Y 546.064,Z 680.363,A -85,B 0,C 180,E1 -3568.881,E2 -3568.881} C_VEL
LIN {X 0,Y 546.16,Z 669.901,A -85,B 0,C 180,E1 -3569.123,E2 -3569.123} C_VEL
LIN {X 0,Y 546.404,Z 619.229,A -85,B 0,C 180,E1 -3569.813,E2 -3569.813} C_VEL
LIN {X 0,Y 546.465,Z 572.849,A -85,B 0,C 180,E1 -3570.427,E2 -3570.427} C_VEL
LIN {X 0,Y 545.022,Z 564.642,A -85,B 0,C 180,E1 -3570.579,E2 -3570.579} C_VEL
LIN {X 0,Y 545.066,Z 562.591,A -85,B 0,C 180,E1 -3571.093,E2 -3571.093} C_VEL
LIN {X 0,Y 545.097,Z 562.584,A -85,B 0,C 180,E1 -3573.175,E2 -3573.175} C_VEL
LIN {X 0,Y 545.043,Z 562.588,A -85,B 0,C 180,E1 -3575.63,E2 -3575.63} C_VEL
LIN {X 0,Y 545.061,Z 562.591,A -85,B 0,C 180,E1 -3578.836,E2 -3578.836} C_VEL
LIN {X 0,Y 545.076,Z 562.585,A -85,B 0,C 180,E1 -3581.195,E2 -3581.195} C_VEL
LIN {X 0,Y 545.067,Z 562.584,A -85,B 0,C 180,E1 -3583.521,E2 -3583.521} C_VEL
LIN {X 0,Y 545.086,Z 562.583,A -85,B 0,C 180,E1 -3585.82,E2 -3585.82} C_VEL
LIN {X 0,Y 545.123,Z 562.582,A -85,B 0,C 180,E1 -3588.849,E2 -3588.849} C_VEL
LIN {X 0,Y 545.127,Z 562.578,A -85,B 0,C 180,E1 -3591.847,E2 -3591.847} C_VEL
LIN {X 0,Y 545.201,Z 562.572,A -85,B 0,C 180,E1 -3594.823,E2 -3594.823} C_VEL
LIN {X 0,Y 545.186,Z 562.569,A -85,B 0,C 180,E1 -3597.784,E2 -3597.784} C_VEL
LIN {X 0,Y 545.206,Z 562.573,A -85,B 0,C 180,E1 -3600.739,E2 -3600.739} C_VEL
LIN {X 0,Y 545.168,Z 562.573,A -85,B 0,C 180,E1 -3602.956,E2 -3602.956} C_VEL
LIN {X 0,Y 545.17,Z 562.573,A -85,B 0,C 180,E1 -3605.92,E2 -3605.92} C_VEL
LIN {X 0,Y 545.119,Z 562.58,A -85,B 0,C 180,E1 -3608.9,E2 -3608.9} C_VEL
LIN {X 0,Y 545.126,Z 562.577,A -85,B 0,C 180,E1 -3611.904,E2 -3611.904} C_VEL
LIN {X 0,Y 545.076,Z 562.585,A -85,B 0,C 180,E1 -3614.944,E2 -3614.944} C_VEL
LIN {X 0,Y 545.075,Z 562.583,A -85,B 0,C 180,E1 -3618.026,E2 -3618.026} C_VEL
LIN {X 0,Y 545.091,Z 562.587,A -85,B 0,C 180,E1 -3620.372,E2 -3620.372} C_VEL
LIN {X 0,Y 545.106,Z 562.578,A -85,B 0,C 180,E1 -3623.558,E2 -3623.558} C_VEL
LIN {X 0,Y 545.081,Z 562.585,A -85,B 0,C 180,E1 -3626.001,E2 -3626.001} C_VEL
LIN {X 0,Y 545.086,Z 562.587,A -85,B 0,C 180,E1 -3628.75,E2 -3628.75} C_VEL
LIN {X 0,Y 545.071,Z 562.583,A -85,B 0,C 180,E1 -3631.683,E2 -3631.683} C_VEL
LIN {X 0,Y 545.078,Z 562.592,A -85,B 0,C 180,E1 -3634.563,E2 -3634.563} C_VEL
LIN {X 0,Y 545.036,Z 562.588,A -85,B 0,C 180,E1 -3637.304,E2 -3637.304} C_VEL
LIN {X 0,Y 545.088,Z 562.585,A -85,B 0,C 180,E1 -3640.141,E2 -3640.141} C_VEL
LIN {X 0,Y 545.083,Z 562.583,A -85,B 0,C 180,E1 -3643.106,E2 -3643.106} C_VEL
LIN {X 0,Y 545.052,Z 562.592,A -85,B 0,C 180,E1 -3646.226,E2 -3646.226} C_VEL
LIN {X 0,Y 545.094,Z 562.584,A -85,B 0,C 180,E1 -3648.888,E2 -3648.888} C_VEL
LIN {X 0,Y 545.085,Z 562.587,A -85,B 0,C 180,E1 -3650.82,E2 -3650.82} C_VEL
LIN {X 0,Y 545.046,Z 562.587,A -85,B 0,C 180,E1 -3653.621,E2 -3653.621} C_VEL
LIN {X 0,Y 545.069,Z 562.592,A -85,B 0,C 180,E1 -3656.329,E2 -3656.329} C_VEL
LIN {X 0,Y 545.065,Z 562.589,A -85,B 0,C 180,E1 -3658.953,E2 -3658.953} C_VEL
LIN {X 0,Y 545.102,Z 562.582,A -85,B 0,C 180,E1 -3661.508,E2 -3661.508} C_VEL
LIN {X 0,Y 545.095,Z 562.616,A -85,B 0,C 180,E1 -3663.847,E2 -3663.847} C_VEL
LIN {X 0,Y 546.822,Z 571.59,A -85,B 0,C 180,E1 -3665.108,E2 -3665.108} C_VEL
LIN {X 0,Y 546.555,Z 590.793,A -85,B 0,C 180,E1 -3667.609,E2 -3667.609} C_VEL
LIN {X 0,Y 546.18,Z 612.754,A -85,B 0,C 180,E1 -3670.455,E2 -3670.455} C_VEL
LIN {X 0,Y 545.743,Z 634.806,A -85,B 0,C 180,E1 -3673.35,E2 -3673.35} C_VEL
LIN {X 0,Y 545.539,Z 650.802,A -85,B 0,C 180,E1 -3675.428,E2 -3675.428} C_VEL
LIN {X 0,Y 546.57,Z 658.889,A -85,B 0,C 180,E1 -3675.569,E2 -3675.569} C_VEL
LIN {X 0,Y 546.269,Z 759.961,A -85,B 0,C 180,E1 -3676.918,E2 -3676.918} C_VEL
LIN {X 0,Y 546.083,Z 772.458,A -85,B 0,C 180,E1 -3677.221,E2 -3677.221} C_VEL
LIN {X 0,Y 545.908,Z 785.371,A -85,B 0,C 180,E1 -3677.689,E2 -3677.689} C_VEL
LIN {X 0,Y 545.73,Z 797.676,A -85,B 0,C 180,E1 -3678.3,E2 -3678.3} C_VEL
LIN {X 0,Y 545.497,Z 809.201,A -85,B 0,C 180,E1 -3679.046,E2 -3679.046} C_VEL
LIN {X 0,Y 545.259,Z 819.606,A -85,B 0,C 180,E1 -3679.886,E2 -3679.886} C_VEL
LIN {X 0,Y 545.084,Z 828.115,A -85,B 0,C 180,E1 -3680.726,E2 -3680.726} C_VEL
LIN {X 0,Y 544.977,Z 835.962,A -85,B 0,C 180,E1 -3681.658,E2 -3681.658} C_VEL
LIN {X 0,Y 544.823,Z 843.623,A -85,B 0,C 180,E1 -3682.775,E2 -3682.775} C_VEL
LIN {X 0,Y 544.776,Z 850.68,A -85,B 0,C 180,E1 -3684.076,E2 -3684.076} C_VEL
LIN {X 0,Y 544.629,Z 855.372,A -85,B 0,C 180,E1 -3685.189,E2 -3685.189} C_VEL
LIN {X 0,Y 544.669,Z 858.96,A -85,B 0,C 180,E1 -3686.301,E2 -3686.301} C_VEL
LIN {X 0,Y 544.651,Z 860.81,A -85,B 0,C 180,E1 -3687.041,E2 -3687.041} C_VEL
LIN {X 0,Y 544.546,Z 863.185,A -85,B 0,C 180,E1 -3688.521,E2 -3688.521} C_VEL
LIN {X 0,Y 544.541,Z 864,A -85,B 0,C 180,E1 -3690,E2 -3690} C_VEL
LIN {X 0,Y 544.546,Z 863.184,A -85,B 0,C 180,E1 -3691.479,E2 -3691.479} C_VEL
LIN {X 0,Y 544.651,Z 860.808,A -85,B 0,C 180,E1 -3692.959,E2 -3692.959} C_VEL
LIN {X 0,Y 544.684,Z 857.895,A -85,B 0,C 180,E1 -3694.069,E2 -3694.069} C_VEL
LIN {X 0,Y 544.654,Z 853.95,A -85,B 0,C 180,E1 -3695.182,E2 -3695.182} C_VEL
LIN {X 0,Y 544.739,Z 848.705,A -85,B 0,C 180,E1 -3696.328,E2 -3696.328} C_VEL
LIN {X 0,Y 544.836,Z 842.468,A -85,B 0,C 180,E1 -3697.411,E2 -3697.411} C_VEL
LIN {X 0,Y 545.006,Z 834.479,A -85,B 0,C 180,E1 -3698.528,E2 -3698.528} C_VEL
LIN {X 0,Y 545.151,Z 826.336,A -85,B 0,C 180,E1 -3699.46,E2 -3699.46} C_VEL
LIN {X 0,Y 545.372,Z 816.403,A -85,B 0,C 180,E1 -3700.394,E2 -3700.394} C_VEL
LIN {X 0,Y 545.566,Z 805.596,A -85,B 0,C 180,E1 -3701.208,E2 -3701.208} C_VEL
LIN {X 0,Y 545.745,Z 794.179,A -85,B 0,C 180,E1 -3701.89,E2 -3701.89} C_VEL
LIN {X 0,Y 545.967,Z 781.99,A -85,B 0,C 180,E1 -3702.451,E2 -3702.451} C_VEL
LIN {X 0,Y 546.123,Z 769.195,A -85,B 0,C 180,E1 -3702.873,E2 -3702.873} C_VEL
LIN {X 0,Y 546.27,Z 755.622,A -85,B 0,C 180,E1 -3703.153,E2 -3703.153} C_VEL
LIN {X 0,Y 546.459,Z 655.868,A -85,B 0,C 180,E1 -3704.475,E2 -3704.475} C_VEL
LIN {X 0,Y 545.64,Z 649.745,A -85,B 0,C 180,E1 -3704.592,E2 -3704.592} C_VEL
LIN {X 0,Y 546.071,Z 623.063,A -85,B 0,C 180,E1 -3707.617,E2 -3707.617} C_VEL
LIN {X 0,Y 546.574,Z 597.801,A -85,B 0,C 180,E1 -3710.511,E2 -3710.511} C_VEL
LIN {X 0,Y 547.009,Z 573.529,A -85,B 0,C 180,E1 -3713.27,E2 -3713.27} C_VEL
LIN {X 0,Y 546.663,Z 569.486,A -85,B 0,C 180,E1 -3713.749,E2 -3713.749} C_VEL
LIN {X 0,Y 545.083,Z 562.587,A -85,B 0,C 180,E1 -3714.621,E2 -3714.621} C_VEL
LIN {X 0,Y 545.097,Z 562.587,A -85,B 0,C 180,E1 -3717.655,E2 -3717.655} C_VEL
LIN {X 0,Y 545.076,Z 562.588,A -85,B 0,C 180,E1 -3720.246,E2 -3720.246} C_VEL
LIN {X 0,Y 545.091,Z 562.581,A -85,B 0,C 180,E1 -3723.064,E2 -3723.064} C_VEL
LIN {X 0,Y 545.061,Z 562.589,A -85,B 0,C 180,E1 -3725.677,E2 -3725.677} C_VEL
LIN {X 0,Y 545.051,Z 562.592,A -85,B 0,C 180,E1 -3728.236,E2 -3728.236} C_VEL
LIN {X 0,Y 545.098,Z 562.579,A -85,B 0,C 180,E1 -3731.112,E2 -3731.112} C_VEL
LIN {X 0,Y 545.055,Z 562.594,A -85,B 0,C 180,E1 -3734.128,E2 -3734.128} C_VEL
LIN {X 0,Y 545.082,Z 562.582,A -85,B 0,C 180,E1 -3736.893,E2 -3736.893} C_VEL
LIN {X 0,Y 545.089,Z 562.585,A -85,B 0,C 180,E1 -3739.859,E2 -3739.859} C_VEL
LIN {X 0,Y 545.073,Z 562.583,A -85,B 0,C 180,E1 -3743.072,E2 -3743.072} C_VEL
LIN {X 0,Y 545.078,Z 562.58,A -85,B 0,C 180,E1 -3745.605,E2 -3745.605} C_VEL
LIN {X 0,Y 545.071,Z 562.593,A -85,B 0,C 180,E1 -3748.317,E2 -3748.317} C_VEL
LIN {X 0,Y 545.084,Z 562.578,A -85,B 0,C 180,E1 -3751.25,E2 -3751.25} C_VEL
LIN {X 0,Y 545.081,Z 562.585,A -85,B 0,C 180,E1 -3753.999,E2 -3753.999} C_VEL
LIN {X 0,Y 545.082,Z 562.587,A -85,B 0,C 180,E1 -3756.441,E2 -3756.441} C_VEL
LIN {X 0,Y 545.089,Z 562.58,A -85,B 0,C 180,E1 -3759.628,E2 -3759.628} C_VEL
LIN {X 0,Y 545.085,Z 562.583,A -85,B 0,C 180,E1 -3762.75,E2 -3762.75} C_VEL
LIN {X 0,Y 545.085,Z 562.58,A -85,B 0,C 180,E1 -3765.82,E2 -3765.82} C_VEL
LIN {X 0,Y 545.123,Z 562.58,A -85,B 0,C 180,E1 -3768.849,E2 -3768.849} C_VEL
LIN {X 0,Y 545.125,Z 562.573,A -85,B 0,C 180,E1 -3771.847,E2 -3771.847} C_VEL
LIN {X 0,Y 545.204,Z 562.573,A -85,B 0,C 180,E1 -3774.823,E2 -3774.823} C_VEL
LIN {X 0,Y 545.186,Z 562.565,A -85,B 0,C 180,E1 -3777.784,E2 -3777.784} C_VEL
LIN {X 0,Y 545.209,Z 562.574,A -85,B 0,C 180,E1 -3780.739,E2 -3780.739} C_VEL
LIN {X 0,Y 545.168,Z 562.576,A -85,B 0,C 180,E1 -3782.956,E2 -3782.956} C_VEL
LIN {X 0,Y 545.169,Z 562.566,A -85,B 0,C 180,E1 -3785.92,E2 -3785.92} C_VEL
LIN {X 0,Y 545.119,Z 562.586,A -85,B 0,C 180,E1 -3788.9,E2 -3788.9} C_VEL
LIN {X 0,Y 545.126,Z 562.573,A -85,B 0,C 180,E1 -3791.904,E2 -3791.904} C_VEL
LIN {X 0,Y 545.075,Z 562.592,A -85,B 0,C 180,E1 -3794.944,E2 -3794.944} C_VEL
LIN {X 0,Y 545.073,Z 562.581,A -85,B 0,C 180,E1 -3798.026,E2 -3798.026} C_VEL
LIN {X 0,Y 545.089,Z 562.581,A -85,B 0,C 180,E1 -3800.372,E2 -3800.372} C_VEL
LIN {X 0,Y 545.083,Z 562.582,A -85,B 0,C 180,E1 -3803.559,E2 -3803.559} C_VEL
LIN {X 0,Y 545.081,Z 562.581,A -85,B 0,C 180,E1 -3806.001,E2 -3806.001} C_VEL
LIN {X 0,Y 545.084,Z 562.586,A -85,B 0,C 180,E1 -3808.75,E2 -3808.75} C_VEL
LIN {X 0,Y 545.07,Z 562.585,A -85,B 0,C 180,E1 -3811.683,E2 -3811.683} C_VEL
LIN {X 0,Y 545.074,Z 562.582,A -85,B 0,C 180,E1 -3814.564,E2 -3814.564} C_VEL
LIN {X 0,Y 545.065,Z 562.59,A -85,B 0,C 180,E1 -3817.023,E2 -3817.023} C_VEL
LIN {X 0,Y 544.388,Z 562.676,A -85,B 0,C 180,E1 -3817.64,E2 -3817.64} C_VEL
LIN {X 0,Y 541.523,Z 563.03,A -85,B 0,C 180,E1 -3818.64,E2 -3818.64} C_VEL
LIN {X 0,Y 539.115,Z 563.33,A -85,B 0,C 180,E1 -3819.446,E2 -3819.446} C_VEL
LIN {X 0,Y 538.093,Z 563.452,A -85,B 0,C 180,E1 -3820.068,E2 -3820.068} C_VEL
LIN {X 0,Y 538.017,Z 563.461,A -85,B 0,C 180,E1 -3820.278,E2 -3820.278} C_VEL
LIN {X 0,Y 538.028,Z 563.458,A -85,B 0,C 180,E1 -3822.989,E2 -3822.989} C_VEL
LIN {X 0,Y 538.016,Z 563.463,A -85,B 0,C 180,E1 -3825.927,E2 -3825.927} C_VEL
LIN {X 0,Y 538.051,Z 563.463,A -85,B 0,C 180,E1 -3829.253,E2 -3829.253} C_VEL
LIN {X 0,Y 537.991,Z 563.464,A -85,B 0,C 180,E1 -3832.123,E2 -3832.123} C_VEL
LIN {X 0,Y 538.018,Z 563.464,A -85,B 0,C 180,E1 -3834.918,E2 -3834.918} C_VEL
LIN {X 0,Y 538.025,Z 563.469,A -85,B 0,C 180,E1 -3837.619,E2 -3837.619} C_VEL
LIN {X 0,Y 538.016,Z 563.464,A -85,B 0,C 180,E1 -3840.24,E2 -3840.24} C_VEL
LIN {X 0,Y 537.996,Z 563.471,A -85,B 0,C 180,E1 -3843.003,E2 -3843.003} C_VEL
LIN {X 0,Y 537.973,Z 564.665,A -85,B 0,C 180,E1 -3843.312,E2 -3843.312} C_VEL
LIN {X 0,Y 539.671,Z 573.81,A -85,B 0,C 180,E1 -3843.491,E2 -3843.491} C_VEL
LIN {X 0,Y 539.281,Z 669.7,A -85,B 0,C 180,E1 -3844.787,E2 -3844.787} C_VEL
LIN {X 0,Y 539.049,Z 682.997,A -85,B 0,C 180,E1 -3845.111,E2 -3845.111} C_VEL
LIN {X 0,Y 538.952,Z 695.988,A -85,B 0,C 180,E1 -3845.6,E2 -3845.6} C_VEL
LIN {X 0,Y 538.718,Z 708.653,A -85,B 0,C 180,E1 -3846.248,E2 -3846.248} C_VEL
LIN {X 0,Y 538.458,Z 719.279,A -85,B 0,C 180,E1 -3846.949,E2 -3846.949} C_VEL
LIN {X 0,Y 538.254,Z 729.075,A -85,B 0,C 180,E1 -3847.75,E2 -3847.75} C_VEL
LIN {X 0,Y 538.011,Z 739.002,A -85,B 0,C 180,E1 -3848.747,E2 -3848.747} C_VEL
LIN {X 0,Y 537.843,Z 747.063,A -85,B 0,C 180,E1 -3849.741,E2 -3849.741} C_VEL
LIN {X 0,Y 537.72,Z 754.832,A -85,B 0,C 180,E1 -3850.929,E2 -3850.929} C_VEL
LIN {X 0,Y 537.644,Z 760.995,A -85,B 0,C 180,E1 -3852.111,E2 -3852.111} C_VEL
LIN {X 0,Y 537.582,Z 765.793,A -85,B 0,C 180,E1 -3853.285,E2 -3853.285} C_VEL
LIN {X 0,Y 537.519,Z 769.387,A -85,B 0,C 180,E1 -3854.453,E2 -3854.453} C_VEL
LIN {X 0,Y 537.51,Z 771.904,A -85,B 0,C 180,E1 -3855.616,E2 -3855.616} C_VEL
LIN {X 0,Y 537.476,Z 773.015,A -85,B 0,C 180,E1 -3856.387,E2 -3856.387} C_VEL
LIN {X 0,Y 537.475,Z 773.697,A -85,B 0,C 180,E1 -3857.157,E2 -3857.157} C_VEL
LIN {X 0,Y 537.47,Z 773.981,A -85,B 0,C 180,E1 -3857.924,E2 -3857.924} C_VEL
LIN {X 0,Y 537.54,Z 773.849,A -85,B 0,C 180,E1 -3858.69,E2 -3858.69} C_VEL
LIN {X 0,Y 537.482,Z 772.316,A -85,B 0,C 180,E1 -3860.213,E2 -3860.213} C_VEL
LIN {X 0,Y 537.474,Z 770.957,A -85,B 0,C 180,E1 -3860.973,E2 -3860.973} C_VEL
LIN {X 0,Y 537.558,Z 768.071,A -85,B 0,C 180,E1 -3862.11,E2 -3862.11} C_VEL
LIN {X 0,Y 537.666,Z 763.41,A -85,B 0,C 180,E1 -3863.425,E2 -3863.425} C_VEL
LIN {X 0,Y 537.638,Z 757.159,A -85,B 0,C 180,E1 -3864.75,E2 -3864.75} C_VEL
LIN {X 0,Y 537.811,Z 750.367,A -85,B 0,C 180,E1 -3865.879,E2 -3865.879} C_VEL
LIN {X 0,Y 537.918,Z 741.914,A -85,B 0,C 180,E1 -3867.004,E2 -3867.004} C_VEL
LIN {X 0,Y 538.155,Z 733.286,A -85,B 0,C 180,E1 -3867.942,E2 -3867.942} C_VEL
LIN {X 0,Y 538.342,Z 722.734,A -85,B 0,C 180,E1 -3868.878,E2 -3868.878} C_VEL
LIN {X 0,Y 538.585,Z 712.17,A -85,B 0,C 180,E1 -3869.626,E2 -3869.626} C_VEL
LIN {X 0,Y 538.888,Z 700.492,A -85,B 0,C 180,E1 -3870.28,E2 -3870.28} C_VEL
LIN {X 0,Y 539.046,Z 688.475,A -85,B 0,C 180,E1 -3870.794,E2 -3870.794} C_VEL
LIN {X 0,Y 539.245,Z 675.051,A -85,B 0,C 180,E1 -3871.19,E2 -3871.19} C_VEL
LIN {X 0,Y 539.337,Z 661.944,A -85,B 0,C 180,E1 -3871.423,E2 -3871.423} C_VEL
LIN {X 0,Y 539.553,Z 572.135,A -85,B 0,C 180,E1 -3872.625,E2 -3872.625} C_VEL
LIN {X 0,Y 538.148,Z 563.77,A -85,B 0,C 180,E1 -3872.784,E2 -3872.784} C_VEL
LIN {X 0,Y 538.148,Z 563.451,A -85,B 0,C 180,E1 -3872.901,E2 -3872.901} C_VEL
LIN {X 0,Y 538.122,Z 563.458,A -85,B 0,C 180,E1 -3875.997,E2 -3875.997} C_VEL
LIN {X 0,Y 538.065,Z 563.463,A -85,B 0,C 180,E1 -3878.261,E2 -3878.261} C_VEL
LIN {X 0,Y 538.12,Z 563.452,A -85,B 0,C 180,E1 -3881.614,E2 -3881.614} C_VEL
LIN {X 0,Y 538.061,Z 563.457,A -85,B 0,C 180,E1 -3884.857,E2 -3884.857} C_VEL
LIN {X 0,Y 538.062,Z 563.459,A -85,B 0,C 180,E1 -3887.54,E2 -3887.54} C_VEL
LIN {X 0,Y 538.041,Z 563.46,A -85,B 0,C 180,E1 -3890.651,E2 -3890.651} C_VEL
LIN {X 0,Y 538.004,Z 563.471,A -85,B 0,C 180,E1 -3893.888,E2 -3893.888} C_VEL
LIN {X 0,Y 538.043,Z 563.464,A -85,B 0,C 180,E1 -3896.366,E2 -3896.366} C_VEL
LIN {X 0,Y 538.034,Z 563.462,A -85,B 0,C 180,E1 -3898.933,E2 -3898.933} C_VEL
LIN {X 0,Y 538.08,Z 563.65,A -85,B 0,C 180,E1 -3901.277,E2 -3901.277} C_VEL
LIN {X 0,Y 538.182,Z 564.544,A -85,B 0,C 180,E1 -3901.325,E2 -3901.325} C_VEL
LIN {X 0,Y 539.687,Z 573.084,A -85,B 0,C 180,E1 -3901.482,E2 -3901.482} C_VEL
LIN {X 0,Y 539.307,Z 668.852,A -85,B 0,C 180,E1 -3902.779,E2 -3902.779} C_VEL
LIN {X 0,Y 539.204,Z 678.593,A -85,B 0,C 180,E1 -3902.995,E2 -3902.995} C_VEL
LIN {X 0,Y 539.016,Z 688.687,A -85,B 0,C 180,E1 -3903.312,E2 -3903.312} C_VEL
LIN {X 0,Y 538.893,Z 698.059,A -85,B 0,C 180,E1 -3903.699,E2 -3903.699} C_VEL
LIN {X 0,Y 538.709,Z 708.063,A -85,B 0,C 180,E1 -3904.222,E2 -3904.222} C_VEL
LIN {X 0,Y 538.526,Z 717.64,A -85,B 0,C 180,E1 -3904.841,E2 -3904.841} C_VEL
LIN {X 0,Y 538.316,Z 726.33,A -85,B 0,C 180,E1 -3905.518,E2 -3905.518} C_VEL
LIN {X 0,Y 538.153,Z 733.964,A -85,B 0,C 180,E1 -3906.223,E2 -3906.223} C_VEL
LIN {X 0,Y 538.002,Z 740.586,A -85,B 0,C 180,E1 -3906.934,E2 -3906.934} C_VEL
LIN {X 0,Y 537.864,Z 748.044,A -85,B 0,C 180,E1 -3907.887,E2 -3907.887} C_VEL
LIN {X 0,Y 537.742,Z 754.332,A -85,B 0,C 180,E1 -3908.853,E2 -3908.853} C_VEL
LIN {X 0,Y 537.686,Z 759.589,A -85,B 0,C 180,E1 -3909.826,E2 -3909.826} C_VEL
LIN {X 0,Y 537.599,Z 763.975,A -85,B 0,C 180,E1 -3910.816,E2 -3910.816} C_VEL
LIN {X 0,Y 537.56,Z 767.547,A -85,B 0,C 180,E1 -3911.823,E2 -3911.823} C_VEL
LIN {X 0,Y 537.488,Z 770.499,A -85,B 0,C 180,E1 -3912.926,E2 -3912.926} C_VEL
LIN {X 0,Y 537.479,Z 772.509,A -85,B 0,C 180,E1 -3914.014,E2 -3914.014} C_VEL
LIN {X 0,Y 537.474,Z 773.654,A -85,B 0,C 180,E1 -3915.081,E2 -3915.081} C_VEL
LIN {X 0,Y 537.461,Z 773.989,A -85,B 0,C 180,E1 -3916.128,E2 -3916.128} C_VEL
LIN {X 0,Y 537.462,Z 773.563,A -85,B 0,C 180,E1 -3917.159,E2 -3917.159} C_VEL
LIN {X 0,Y 537.494,Z 772.374,A -85,B 0,C 180,E1 -3918.183,E2 -3918.183} C_VEL
LIN {X 0,Y 537.485,Z 770.174,A -85,B 0,C 180,E1 -3919.321,E2 -3919.321} C_VEL
LIN {X 0,Y 537.59,Z 765.732,A -85,B 0,C 180,E1 -3920.808,E2 -3920.808} C_VEL
LIN {X 0,Y 537.625,Z 761.422,A -85,B 0,C 180,E1 -3921.877,E2 -3921.877} C_VEL
LIN {X 0,Y 537.673,Z 756.426,A -85,B 0,C 180,E1 -3922.875,E2 -3922.875} C_VEL
LIN {X 0,Y 537.783,Z 751.201,A -85,B 0,C 180,E1 -3923.747,E2 -3923.747} C_VEL
LIN {X 0,Y 537.896,Z 744.521,A -85,B 0,C 180,E1 -3924.679,E2 -3924.679} C_VEL
LIN {X 0,Y 538.084,Z 736.531,A -85,B 0,C 180,E1 -3925.604,E2 -3925.604} C_VEL
LIN {X 0,Y 538.254,Z 728.372,A -85,B 0,C 180,E1 -3926.396,E2 -3926.396} C_VEL
LIN {X 0,Y 538.437,Z 719.854,A -85,B 0,C 180,E1 -3927.09,E2 -3927.09} C_VEL
LIN {X 0,Y 538.638,Z 711.569,A -85,B 0,C 180,E1 -3927.659,E2 -3927.659} C_VEL
LIN {X 0,Y 538.794,Z 701.624,A -85,B 0,C 180,E1 -3928.22,E2 -3928.22} C_VEL
LIN {X 0,Y 538.971,Z 691.682,A -85,B 0,C 180,E1 -3928.666,E2 -3928.666} C_VEL
LIN {X 0,Y 539.142,Z 680.893,A -85,B 0,C 180,E1 -3929.033,E2 -3929.033} C_VEL
LIN {X 0,Y 539.238,Z 670.289,A -85,B 0,C 180,E1 -3929.286,E2 -3929.286} C_VEL
LIN {X 0,Y 539.428,Z 637.762,A -85,B 0,C 180,E1 -3929.745,E2 -3929.745} C_VEL
LIN {X 0,Y 539.604,Z 573.653,A -85,B 0,C 180,E1 -3930.603,E2 -3930.603} C_VEL
LIN {X 0,Y 537.998,Z 564.651,A -85,B 0,C 180,E1 -3930.785,E2 -3930.785} C_VEL
LIN {X 0,Y 538.009,Z 563.47,A -85,B 0,C 180,E1 -3931.097,E2 -3931.097} C_VEL
LIN {X 0,Y 538.042,Z 563.462,A -85,B 0,C 180,E1 -3933.633,E2 -3933.633} C_VEL
LIN {X 0,Y 538.014,Z 563.467,A -85,B 0,C 180,E1 -3936.117,E2 -3936.117} C_VEL
LIN {X 0,Y 538.034,Z 563.461,A -85,B 0,C 180,E1 -3939.348,E2 -3939.348} C_VEL
LIN {X 0,Y 538.063,Z 563.466,A -85,B 0,C 180,E1 -3942.517,E2 -3942.517} C_VEL
LIN {X 0,Y 538.054,Z 563.458,A -85,B 0,C 180,E1 -3945.63,E2 -3945.63} C_VEL
LIN {X 0,Y 538.08,Z 563.462,A -85,B 0,C 180,E1 -3948.702,E2 -3948.702} C_VEL
LIN {X 0,Y 538.083,Z 563.455,A -85,B 0,C 180,E1 -3951.74,E2 -3951.74} C_VEL
LIN {X 0,Y 538.177,Z 563.448,A -85,B 0,C 180,E1 -3954.755,E2 -3954.755} C_VEL
LIN {X 0,Y 538.158,Z 563.444,A -85,B 0,C 180,E1 -3957.755,E2 -3957.755} C_VEL
LIN {X 0,Y 538.176,Z 563.448,A -85,B 0,C 180,E1 -3960.748,E2 -3960.748} C_VEL
LIN {X 0,Y 538.134,Z 563.449,A -85,B 0,C 180,E1 -3962.994,E2 -3962.994} C_VEL
LIN {X 0,Y 538.123,Z 563.451,A -85,B 0,C 180,E1 -3965.997,E2 -3965.997} C_VEL
LIN {X 0,Y 538.068,Z 563.457,A -85,B 0,C 180,E1 -3969.018,E2 -3969.018} C_VEL
LIN {X 0,Y 538.074,Z 563.457,A -85,B 0,C 180,E1 -3972.063,E2 -3972.063} C_VEL
LIN {X 0,Y 538.036,Z 563.46,A -85,B 0,C 180,E1 -3975.144,E2 -3975.144} C_VEL
LIN {X 0,Y 538.027,Z 563.464,A -85,B 0,C 180,E1 -3978.27,E2 -3978.27} C_VEL
LIN {X 0,Y 538.034,Z 563.466,A -85,B 0,C 180,E1 -3980.652,E2 -3980.652} C_VEL
LIN {X 0,Y 538.033,Z 563.46,A -85,B 0,C 180,E1 -3983.887,E2 -3983.887} C_VEL
LIN {X 0,Y 538.043,Z 563.466,A -85,B 0,C 180,E1 -3986.367,E2 -3986.367} C_VEL
LIN {X 0,Y 538.048,Z 563.461,A -85,B 0,C 180,E1 -3988.939,E2 -3988.939} C_VEL
LIN {X 0,Y 538.021,Z 563.463,A -85,B 0,C 180,E1 -3991.891,E2 -3991.891} C_VEL
LIN {X 0,Y 538.027,Z 563.469,A -85,B 0,C 180,E1 -3994.622,E2 -3994.622} C_VEL
LIN {X 0,Y 538.004,Z 563.465,A -85,B 0,C 180,E1 -3997.172,E2 -3997.172} C_VEL
LIN {X 0,Y 538.049,Z 563.458,A -85,B 0,C 180,E1 -3999.795,E2 -3999.795} C_VEL
LIN {X 0,Y 538.02,Z 563.467,A -85,B 0,C 180,E1 -4002.786,E2 -4002.786} C_VEL
LIN {X 0,Y 538.027,Z 563.463,A -85,B 0,C 180,E1 -4005.141,E2 -4005.141} C_VEL
LIN {X 0,Y 538.037,Z 563.466,A -85,B 0,C 180,E1 -4008.229,E2 -4008.229} C_VEL
LIN {X 0,Y 538.015,Z 563.464,A -85,B 0,C 180,E1 -4011.171,E2 -4011.171} C_VEL
LIN {X 0,Y 537.999,Z 563.469,A -85,B 0,C 180,E1 -4014.088,E2 -4014.088} C_VEL
LIN {X 0,Y 538.03,Z 563.467,A -85,B 0,C 180,E1 -4016.728,E2 -4016.728} C_VEL
LIN {X 0,Y 538.025,Z 563.463,A -85,B 0,C 180,E1 -4019.557,E2 -4019.557} C_VEL
LIN {X 0,Y 538.044,Z 563.464,A -85,B 0,C 180,E1 -4021.951,E2 -4021.951} C_VEL
LIN {X 0,Y 538.086,Z 563.598,A -85,B 0,C 180,E1 -4023.701,E2 -4023.701} C_VEL
LIN {X 0,Y 539.85,Z 572.464,A -85,B 0,C 180,E1 -4024.97,E2 -4024.97} C_VEL
LIN {X 0,Y 539.648,Z 589.384,A -85,B 0,C 180,E1 -4027.209,E2 -4027.209} C_VEL
LIN {X 0,Y 539.216,Z 612.273,A -85,B 0,C 180,E1 -4030.192,E2 -4030.192} C_VEL
LIN {X 0,Y 538.836,Z 633.336,A -85,B 0,C 180,E1 -4032.935,E2 -4032.935} C_VEL
LIN {X 0,Y 538.544,Z 650.833,A -85,B 0,C 180,E1 -4035.239,E2 -4035.239} C_VEL
LIN {X 0,Y 539.7,Z 659.772,A -85,B 0,C 180,E1 -4035.393,E2 -4035.393} C_VEL
LIN {X 0,Y 539.371,Z 759.96,A -85,B 0,C 180,E1 -4036.748,E2 -4036.748} C_VEL
LIN {X 0,Y 539.159,Z 772.457,A -85,B 0,C 180,E1 -4037.054,E2 -4037.054} C_VEL
LIN {X 0,Y 538.962,Z 785.37,A -85,B 0,C 180,E1 -4037.528,E2 -4037.528} C_VEL
LIN {X 0,Y 538.787,Z 797.201,A -85,B 0,C 180,E1 -4038.119,E2 -4038.119} C_VEL
LIN {X 0,Y 538.511,Z 809.2,A -85,B 0,C 180,E1 -4038.902,E2 -4038.902} C_VEL
LIN {X 0,Y 538.262,Z 819.607,A -85,B 0,C 180,E1 -4039.753,E2 -4039.753} C_VEL
LIN {X 0,Y 538.066,Z 828.116,A -85,B 0,C 180,E1 -4040.604,E2 -4040.604} C_VEL
LIN {X 0,Y 537.921,Z 835.962,A -85,B 0,C 180,E1 -4041.548,E2 -4041.548} C_VEL
LIN {X 0,Y 537.754,Z 843.623,A -85,B 0,C 180,E1 -4042.679,E2 -4042.679} C_VEL
LIN {X 0,Y 537.693,Z 850.68,A -85,B 0,C 180,E1 -4043.998,E2 -4043.998} C_VEL
LIN {X 0,Y 537.54,Z 855.372,A -85,B 0,C 180,E1 -4045.125,E2 -4045.125} C_VEL
LIN {X 0,Y 537.591,Z 858.961,A -85,B 0,C 180,E1 -4046.252,E2 -4046.252} C_VEL
LIN {X 0,Y 537.551,Z 860.81,A -85,B 0,C 180,E1 -4047.002,E2 -4047.002} C_VEL
LIN {X 0,Y 537.451,Z 863.185,A -85,B 0,C 180,E1 -4048.501,E2 -4048.501} C_VEL
LIN {X 0,Y 537.442,Z 864,A -85,B 0,C 180,E1 -4050,E2 -4050} C_VEL
LIN {X 0,Y 537.451,Z 863.183,A -85,B 0,C 180,E1 -4051.499,E2 -4051.499} C_VEL
LIN {X 0,Y 537.551,Z 860.807,A -85,B 0,C 180,E1 -4052.998,E2 -4052.998} C_VEL
LIN {X 0,Y 537.603,Z 857.895,A -85,B 0,C 180,E1 -4054.123,E2 -4054.123} C_VEL
LIN {X 0,Y 537.588,Z 853.95,A -85,B 0,C 180,E1 -4055.25,E2 -4055.25} C_VEL
LIN {X 0,Y 537.65,Z 849.081,A -85,B 0,C 180,E1 -4056.335,E2 -4056.335} C_VEL
LIN {X 0,Y 537.79,Z 842.468,A -85,B 0,C 180,E1 -4057.509,E2 -4057.509} C_VEL
LIN {X 0,Y 537.972,Z 834.479,A -85,B 0,C 180,E1 -4058.64,E2 -4058.64} C_VEL
LIN {X 0,Y 538.142,Z 826.336,A -85,B 0,C 180,E1 -4059.585,E2 -4059.585} C_VEL
LIN {X 0,Y 538.374,Z 816.402,A -85,B 0,C 180,E1 -4060.53,E2 -4060.53} C_VEL
LIN {X 0,Y 538.576,Z 806.593,A -85,B 0,C 180,E1 -4061.288,E2 -4061.288} C_VEL
LIN {X 0,Y 538.747,Z 795.851,A -85,B 0,C 180,E1 -4061.957,E2 -4061.957} C_VEL
LIN {X 0,Y 538.993,Z 783.119,A -85,B 0,C 180,E1 -4062.567,E2 -4062.567} C_VEL
LIN {X 0,Y 539.209,Z 770.108,A -85,B 0,C 180,E1 -4063.017,E2 -4063.017} C_VEL
LIN {X 0,Y 539.369,Z 757.126,A -85,B 0,C 180,E1 -4063.3,E2 -4063.3} C_VEL
LIN {X 0,Y 539.541,Z 656.073,A -85,B 0,C 180,E1 -4064.662,E2 -4064.662} C_VEL
LIN {X 0,Y 538.692,Z 649.729,A -85,B 0,C 180,E1 -4064.786,E2 -4064.786} C_VEL
LIN {X 0,Y 539.243,Z 620.757,A -85,B 0,C 180,E1 -4068.111,E2 -4068.111} C_VEL
LIN {X 0,Y 539.747,Z 593.815,A -85,B 0,C 180,E1 -4071.181,E2 -4071.181} C_VEL
LIN {X 0,Y 540.111,Z 572.995,A -85,B 0,C 180,E1 -4073.585,E2 -4073.585} C_VEL
LIN {X 0,Y 538.068,Z 563.461,A -85,B 0,C 180,E1 -4074.809,E2 -4074.809} C_VEL
LIN {X 0,Y 538.066,Z 563.461,A -85,B 0,C 180,E1 -4077.353,E2 -4077.353} C_VEL
LIN {X 0,Y 538.017,Z 563.47,A -85,B 0,C 180,E1 -4079.76,E2 -4079.76} C_VEL
LIN {X 0,Y 538.026,Z 563.465,A -85,B 0,C 180,E1 -4082.381,E2 -4082.381} C_VEL
LIN {X 0,Y 538.02,Z 563.462,A -85,B 0,C 180,E1 -4085.082,E2 -4085.082} C_VEL
LIN {X 0,Y 537.991,Z 563.473,A -85,B 0,C 180,E1 -4087.877,E2 -4087.877} C_VEL
LIN {X 0,Y 538.075,Z 563.455,A -85,B 0,C 180,E1 -4090.772,E2 -4090.772} C_VEL
LIN {X 0,Y 538.026,Z 563.47,A -85,B 0,C 180,E1 -4094.074,E2 -4094.074} C_VEL
LIN {X 0,Y 538.019,Z 563.461,A -85,B 0,C 180,E1 -4097.214,E2 -4097.214} C_VEL
LIN {X 0,Y 538.05,Z 563.464,A -85,B 0,C 180,E1 -4100.205,E2 -4100.205} C_VEL
LIN {X 0,Y 538.027,Z 563.461,A -85,B 0,C 180,E1 -4103.067,E2 -4103.067} C_VEL
LIN {X 0,Y 538.02,Z 563.461,A -85,B 0,C 180,E1 -4105.827,E2 -4105.827} C_VEL
LIN {X 0,Y 538.017,Z 563.468,A -85,B 0,C 180,E1 -4108.499,E2 -4108.499} C_VEL
LIN {X 0,Y 538.051,Z 563.454,A -85,B 0,C 180,E1 -4111.099,E2 -4111.099} C_VEL
LIN {X 0,Y 538.043,Z 563.459,A -85,B 0,C 180,E1 -4113.633,E2 -4113.633} C_VEL
LIN {X 0,Y 538.014,Z 563.467,A -85,B 0,C 180,E1 -4116.117,E2 -4116.117} C_VEL
LIN {X 0,Y 538.033,Z 563.459,A -85,B 0,C 180,E1 -4119.348,E2 -4119.348} C_VEL
LIN {X 0,Y 538.063,Z 563.462,A -85,B 0,C 180,E1 -4122.517,E2 -4122.517} C_VEL
LIN {X 0,Y 538.054,Z 563.455,A -85,B 0,C 180,E1 -4125.63,E2 -4125.63} C_VEL
LIN {X 0,Y 538.08,Z 563.46,A -85,B 0,C 180,E1 -4128.702,E2 -4128.702} C_VEL
LIN {X 0,Y 538.081,Z 563.449,A -85,B 0,C 180,E1 -4131.739,E2 -4131.739} C_VEL
LIN {X 0,Y 538.18,Z 563.449,A -85,B 0,C 180,E1 -4134.755,E2 -4134.755} C_VEL
LIN {X 0,Y 538.158,Z 563.44,A -85,B 0,C 180,E1 -4137.755,E2 -4137.755} C_VEL
LIN {X 0,Y 538.178,Z 563.45,A -85,B 0,C 180,E1 -4140.748,E2 -4140.748} C_VEL
LIN {X 0,Y 538.134,Z 563.452,A -85,B 0,C 180,E1 -4142.994,E2 -4142.994} C_VEL
LIN {X 0,Y 538.123,Z 563.444,A -85,B 0,C 180,E1 -4145.997,E2 -4145.997} C_VEL
LIN {X 0,Y 538.068,Z 563.462,A -85,B 0,C 180,E1 -4149.018,E2 -4149.018} C_VEL
LIN {X 0,Y 538.074,Z 563.452,A -85,B 0,C 180,E1 -4152.063,E2 -4152.063} C_VEL
LIN {X 0,Y 538.035,Z 563.466,A -85,B 0,C 180,E1 -4155.144,E2 -4155.144} C_VEL
LIN {X 0,Y 538.026,Z 563.459,A -85,B 0,C 180,E1 -4158.27,E2 -4158.27} C_VEL
LIN {X 0,Y 538.033,Z 563.462,A -85,B 0,C 180,E1 -4160.652,E2 -4160.652} C_VEL
LIN {X 0,Y 538.015,Z 563.46,A -85,B 0,C 180,E1 -4163.888,E2 -4163.888} C_VEL
LIN {X 0,Y 538.042,Z 563.459,A -85,B 0,C 180,E1 -4166.367,E2 -4166.367} C_VEL
LIN {X 0,Y 538.048,Z 563.465,A -85,B 0,C 180,E1 -4168.939,E2 -4168.939} C_VEL
LIN {X 0,Y 538.02,Z 563.462,A -85,B 0,C 180,E1 -4171.891,E2 -4171.891} C_VEL
LIN {X 0,Y 538.024,Z 563.461,A -85,B 0,C 180,E1 -4174.621,E2 -4174.621} C_VEL
LIN {X 0,Y 538.018,Z 563.471,A -85,B 0,C 180,E1 -4177.174,E2 -4177.174} C_VEL
LIN {X 0,Y 538.017,Z 563.461,A -85,B 0,C 180,E1 -4180.278,E2 -4180.278} C_VEL
LIN {X 0,Y 537.367,Z 563.546,A -85,B 0,C 180,E1 -4180.904,E2 -4180.904} C_VEL
LIN {X 0,Y 534.518,Z 563.907,A -85,B 0,C 180,E1 -4181.919,E2 -4181.919} C_VEL
LIN {X 0,Y 532.094,Z 564.211,A -85,B 0,C 180,E1 -4182.736,E2 -4182.736} C_VEL
LIN {X 0,Y 531.047,Z 564.338,A -85,B 0,C 180,E1 -4183.367,E2 -4183.367} C_VEL
LIN {X 0,Y 530.959,Z 564.346,A -85,B 0,C 180,E1 -4183.581,E2 -4183.581} C_VEL
LIN {X 0,Y 530.95,Z 564.342,A -85,B 0,C 180,E1 -4186.505,E2 -4186.505} C_VEL
LIN {X 0,Y 530.985,Z 564.339,A -85,B 0,C 180,E1 -4188.977,E2 -4188.977} C_VEL
LIN {X 0,Y 530.956,Z 564.345,A -85,B 0,C 180,E1 -4191.53,E2 -4191.53} C_VEL
LIN {X 0,Y 530.98,Z 564.339,A -85,B 0,C 180,E1 -4194.383,E2 -4194.383} C_VEL
LIN {X 0,Y 530.969,Z 564.345,A -85,B 0,C 180,E1 -4197.134,E2 -4197.134} C_VEL
LIN {X 0,Y 530.969,Z 564.346,A -85,B 0,C 180,E1 -4199.804,E2 -4199.804} C_VEL
LIN {X 0,Y 531.01,Z 564.34,A -85,B 0,C 180,E1 -4202.832,E2 -4202.832} C_VEL
LIN {X 0,Y 530.983,Z 564.406,A -85,B 0,C 180,E1 -4202.937,E2 -4202.937} C_VEL
LIN {X 0,Y 530.978,Z 565.174,A -85,B 0,C 180,E1 -4203.123,E2 -4203.123} C_VEL
LIN {X 0,Y 532.778,Z 574.615,A -85,B 0,C 180,E1 -4203.305,E2 -4203.305} C_VEL
LIN {X 0,Y 532.384,Z 670.295,A -85,B 0,C 180,E1 -4204.621,E2 -4204.621} C_VEL
LIN {X 0,Y 532.153,Z 683.437,A -85,B 0,C 180,E1 -4204.949,E2 -4204.949} C_VEL
LIN {X 0,Y 532.034,Z 695.58,A -85,B 0,C 180,E1 -4205.412,E2 -4205.412} C_VEL
LIN {X 0,Y 531.791,Z 707.492,A -85,B 0,C 180,E1 -4206.023,E2 -4206.023} C_VEL
LIN {X 0,Y 531.529,Z 718.359,A -85,B 0,C 180,E1 -4206.734,E2 -4206.734} C_VEL
LIN {X 0,Y 531.241,Z 728.556,A -85,B 0,C 180,E1 -4207.565,E2 -4207.565} C_VEL
LIN {X 0,Y 531.038,Z 737.475,A -85,B 0,C 180,E1 -4208.454,E2 -4208.454} C_VEL
LIN {X 0,Y 530.836,Z 745.797,A -85,B 0,C 180,E1 -4209.461,E2 -4209.461} C_VEL
LIN {X 0,Y 530.697,Z 753.871,A -85,B 0,C 180,E1 -4210.667,E2 -4210.667} C_VEL
LIN {X 0,Y 530.584,Z 760.219,A -85,B 0,C 180,E1 -4211.864,E2 -4211.864} C_VEL
LIN {X 0,Y 530.5,Z 765.185,A -85,B 0,C 180,E1 -4213.055,E2 -4213.055} C_VEL
LIN {X 0,Y 530.454,Z 768.936,A -85,B 0,C 180,E1 -4214.241,E2 -4214.241} C_VEL
LIN {X 0,Y 530.42,Z 771.597,A -85,B 0,C 180,E1 -4215.419,E2 -4215.419} C_VEL
LIN {X 0,Y 530.403,Z 772.828,A -85,B 0,C 180,E1 -4216.202,E2 -4216.202} C_VEL
LIN {X 0,Y 530.368,Z 773.595,A -85,B 0,C 180,E1 -4216.982,E2 -4216.982} C_VEL
LIN {X 0,Y 530.381,Z 773.947,A -85,B 0,C 180,E1 -4217.76,E2 -4217.76} C_VEL
LIN {X 0,Y 530.448,Z 773.874,A -85,B 0,C 180,E1 -4218.65,E2 -4218.65} C_VEL
